  MoveL 2000 to (240.59, 49.33, 41.04) mm, rotated rx -180 ry 0 rz 180 deg; joints [-31.47, 47.148, -71.346, 33.863, 110.463, 13.203]
  Call Extruder(203.73378)
  MoveL 2001 to (240.64, 49.63, 41.04) mm, rotated rx -180 ry 0 rz 180 deg; joints [-31.612, 47.167, -71.344, 34.007, 110.413, 13.242]
  MoveL 2002 to (240.64, 49.63, 41.04) mm, rotated rx -180 ry 0 rz 180 deg; joints [-31.612, 47.167, -71.344, 34.007, 110.413, 13.242]
  Call Extruder(203.89480)
  MoveL 2003 to (240.69, 49.94, 41.04) mm, rotated rx 180 ry 0 rz 180 deg; joints [-31.755, 47.186, -71.343, 34.15, 110.364, 13.281]
  MoveL 2004 to (240.69, 49.94, 41.04) mm, rotated rx 180 ry 0 rz 180 deg; joints [-31.755, 47.186, -71.343, 34.15, 110.364, 13.281]
  Call Extruder(204.05509)
  MoveL 2005 to (240.74, 50.24, 41.04) mm, rotated rx 180 ry 0 rz 180 deg; joints [-31.895, 47.205, -71.341, 34.292, 110.314, 13.32]
  MoveL 2006 to (240.74, 50.24, 41.04) mm, rotated rx 180 ry 0 rz 180 deg; joints [-31.895, 47.205, -71.341, 34.292, 110.314, 13.32]
  Call Extruder(204.21465)
  MoveL 2007 to (240.78, 50.55, 41.04) mm, rotated rx 180 ry 0 rz 180 deg; joints [-32.036, 47.224, -71.34, 34.434, 110.265, 13.358]
  MoveL 2008 to (240.78, 50.55, 41.04) mm, rotated rx 180 ry 0 rz 180 deg; joints [-32.036, 47.224, -71.34, 34.434, 110.265, 13.358]
  Call Extruder(204.37349)
  MoveL 2009 to (240.83, 50.86, 41.04) mm, rotated rx -180 ry 0 rz 180 deg; joints [-32.176, 47.243, -71.338, 34.575, 110.215, 13.396]
  MoveL 2010 to (240.83, 50.86, 41.04) mm, rotated rx -180 ry 0 rz 180 deg; joints [-32.176, 47.243, -71.338, 34.575, 110.215, 13.396]
  Call Extruder(204.55216)
  MoveL 2011 to (240.88, 51.2, 41.04) mm, rotated rx 180 ry 0 rz -180 deg; joints [-32.337, 47.264, -71.336, 34.736, 110.159, 13.439]
  MoveL 2012 to (240.88, 51.2, 41.04) mm, rotated rx 180 ry 0 rz -180 deg; joints [-32.337, 47.264, -71.336, 34.736, 110.159, 13.439]
  Call Extruder(204.75060)
  MoveL 2013 to (240.92, 51.59, 41.04) mm, rotated rx -180 ry 0 rz 180 deg; joints [-32.518, 47.288, -71.334, 34.918, 110.096, 13.488]
  MoveL 2014 to (240.92, 51.59, 41.04) mm, rotated rx -180 ry 0 rz 180 deg; joints [-32.518, 47.288, -71.334, 34.918, 110.096, 13.488]
  Call Extruder(204.94818)
  MoveL 2015 to (240.97, 51.98, 41.04) mm, rotated rx 180 ry 0 rz 180 deg; joints [-32.697, 47.311, -71.332, 35.099, 110.034, 13.537]
  MoveL 2016 to (240.97, 51.98, 41.04) mm, rotated rx 180 ry 0 rz 180 deg; joints [-32.697, 47.311, -71.332, 35.099, 110.034, 13.537]
  Call Extruder(205.14488)
  MoveL 2017 to (241.02, 52.37, 41.04) mm, rotated rx -180 ry 0 rz 180 deg; joints [-32.876, 47.334, -71.33, 35.279, 109.971, 13.584]
  MoveL 2018 to (241.02, 52.37, 41.04) mm, rotated rx -180 ry 0 rz 180 deg; joints [-32.876, 47.334, -71.33, 35.279, 109.971, 13.584]
  Call Extruder(205.34072)
  MoveL 2019 to (241.06, 52.75, 41.04) mm, rotated rx 180 ry 0 rz 180 deg; joints [-33.055, 47.357, -71.328, 35.458, 109.908, 13.632]
  MoveL 2020 to (241.06, 52.75, 41.04) mm, rotated rx 180 ry 0 rz 180 deg; joints [-33.055, 47.357, -71.328, 35.458, 109.908, 13.632]
  Call Extruder(205.63616)
  MoveL 2021 to (241.11, 53.34, 41.04) mm, rotated rx -180 ry 0 rz 180 deg; joints [-33.331, 47.391, -71.325, 35.736, 109.813, 13.706]
  MoveL 2022 to (241.11, 53.34, 41.04) mm, rotated rx -180 ry 0 rz 180 deg; joints [-33.331, 47.391, -71.325, 35.736, 109.813, 13.706]
  Call Extruder(205.93027)
  MoveL 2023 to (241.16, 53.93, 41.04) mm, rotated rx 180 ry 0 rz 180 deg; joints [-33.606, 47.426, -71.322, 36.012, 109.717, 13.779]
  MoveL 2024 to (241.16, 53.93, 41.04) mm, rotated rx 180 ry 0 rz 180 deg; joints [-33.606, 47.426, -71.322, 36.012, 109.717, 13.779]
  Call Extruder(206.22304)
  MoveL 2025 to (241.2, 54.52, 41.04) mm, rotated rx -180 ry 0 rz 180 deg; joints [-33.878, 47.46, -71.319, 36.285, 109.622, 13.85]
  MoveL 2026 to (241.2, 54.52, 41.04) mm, rotated rx -180 ry 0 rz 180 deg; joints [-33.878, 47.46, -71.319, 36.285, 109.622, 13.85]
  Call Extruder(206.79649)
  MoveL 2027 to (241.25, 55.68, 41.04) mm, rotated rx 180 ry 0 rz 180 deg; joints [-34.425, 47.525, -71.313, 36.832, 109.434, 13.993]
  MoveL 2028 to (241.25, 55.68, 41.04) mm, rotated rx 180 ry 0 rz 180 deg; joints [-34.425, 47.525, -71.313, 36.832, 109.434, 13.993]
  Call Extruder(207.51032)
  MoveL 2029 to (241.29, 57.14, 41.04) mm, rotated rx 180 ry 0 rz 180 deg; joints [-35.104, 47.605, -71.305, 37.512, 109.198, 14.167]
  Call Extruder(249.57521)
  MoveL 2030 to (241.29, 142.86, 41.03) mm, rotated rx 180 ry 0 rz 180 deg; joints [-60.361, 53.167, -69.896, 61.414, 98.184, 14.641]
  Call Extruder(250.00364)
  MoveL 2031 to (241.27, 143.73, 41.04) mm, rotated rx -180 ry 0 rz 180 deg; joints [-60.516, 53.225, -69.87, 61.555, 98.105, 14.588]
  MoveL 2032 to (241.27, 143.73, 41.04) mm, rotated rx -180 ry 0 rz 180 deg; joints [-60.516, 53.225, -69.87, 61.555, 98.105, 14.588]
  Call Extruder(250.57709)
  MoveL 2033 to (241.23, 144.9, 41.04) mm, rotated rx 180 ry 0 rz 180 deg; joints [-60.726, 53.301, -69.836, 61.747, 97.999, 14.519]
  MoveL 2034 to (241.23, 144.9, 41.04) mm, rotated rx 180 ry 0 rz 180 deg; joints [-60.726, 53.301, -69.836, 61.747, 97.999, 14.519]
  Call Extruder(251.01142)
  MoveL 2035 to (241.18, 145.77, 41.04) mm, rotated rx 180 ry 0 rz 180 deg; joints [-60.887, 53.358, -69.81, 61.894, 97.92, 14.467]
  MoveL 2036 to (241.18, 145.77, 41.04) mm, rotated rx 180 ry 0 rz 180 deg; joints [-60.887, 53.358, -69.81, 61.894, 97.92, 14.467]
  Call Extruder(251.30553)
  MoveL 2037 to (241.13, 146.36, 41.04) mm, rotated rx -180 ry 0 rz 180 deg; joints [-61, 53.396, -69.793, 61.997, 97.866, 14.433]
  MoveL 2038 to (241.13, 146.36, 41.04) mm, rotated rx -180 ry 0 rz 180 deg; joints [-61, 53.396, -69.793, 61.997, 97.866, 14.433]
  Call Extruder(251.60097)
  MoveL 2039 to (241.09, 146.95, 41.04) mm, rotated rx -180 ry 0 rz 180 deg; joints [-61.111, 53.434, -69.775, 62.099, 97.813, 14.398]
  MoveL 2040 to (241.09, 146.95, 41.04) mm, rotated rx -180 ry 0 rz 180 deg; joints [-61.111, 53.434, -69.775, 62.099, 97.813, 14.398]
  Call Extruder(251.84723)
  MoveL 2041 to (241.04, 147.44, 41.04) mm, rotated rx 180 ry 0 rz 180 deg; joints [-61.205, 53.465, -69.761, 62.186, 97.768, 14.37]
  MoveL 2042 to (241.04, 147.44, 41.04) mm, rotated rx 180 ry 0 rz 180 deg; joints [-61.205, 53.465, -69.761, 62.186, 97.768, 14.37]
  Call Extruder(252.04393)
  MoveL 2043 to (240.99, 147.83, 41.04) mm, rotated rx 180 ry 0 rz 180 deg; joints [-61.282, 53.489, -69.75, 62.257, 97.732, 14.349]
  MoveL 2044 to (240.99, 147.83, 41.04) mm, rotated rx 180 ry 0 rz 180 deg; joints [-61.282, 53.489, -69.75, 62.257, 97.732, 14.349]
  Call Extruder(252.24151)
  MoveL 2045 to (240.95, 148.22, 41.04) mm, rotated rx -180 ry 0 rz 180 deg; joints [-61.359, 53.513, -69.738, 62.328, 97.697, 14.327]
  MoveL 2046 to (240.95, 148.22, 41.04) mm, rotated rx -180 ry 0 rz 180 deg; joints [-61.359, 53.513, -69.738, 62.328, 97.697, 14.327]
  Call Extruder(252.43995)
  MoveL 2047 to (240.9, 148.6, 41.04) mm, rotated rx -180 ry 0 rz 180 deg; joints [-61.436, 53.537, -69.727, 62.398, 97.661, 14.305]
  MoveL 2048 to (240.9, 148.6, 41.04) mm, rotated rx -180 ry 0 rz 180 deg; joints [-61.436, 53.537, -69.727, 62.398, 97.661, 14.305]
  Call Extruder(252.63926)
  MoveL 2049 to (240.86, 148.99, 41.04) mm, rotated rx 180 ry 0 rz 180 deg; joints [-61.512, 53.562, -69.715, 62.469, 97.626, 14.283]
  MoveL 2050 to (240.86, 148.99, 41.04) mm, rotated rx 180 ry 0 rz 180 deg; joints [-61.512, 53.562, -69.715, 62.469, 97.626, 14.283]
  Call Extruder(252.79809)
  MoveL 2051 to (240.81, 149.3, 41.04) mm, rotated rx -180 ry 0 rz 180 deg; joints [-61.575, 53.58, -69.707, 62.527, 97.597, 14.266]
  MoveL 2052 to (240.81, 149.3, 41.04) mm, rotated rx -180 ry 0 rz 180 deg; joints [-61.575, 53.58, -69.707, 62.527, 97.597, 14.266]
  Call Extruder(252.95765)
  MoveL 2053 to (240.76, 149.6, 41.04) mm, rotated rx 180 ry 0 rz 180 deg; joints [-61.639, 53.599, -69.698, 62.586, 97.569, 14.25]
  MoveL 2054 to (240.76, 149.6, 41.04) mm, rotated rx 180 ry 0 rz 180 deg; joints [-61.639, 53.599, -69.698, 62.586, 97.569, 14.25]
  Call Extruder(253.11794)
  MoveL 2055 to (240.71, 149.91, 41.04) mm, rotated rx -180 ry 0 rz 180 deg; joints [-61.702, 53.618, -69.689, 62.645, 97.541, 14.233]
  MoveL 2056 to (240.71, 149.91, 41.04) mm, rotated rx -180 ry 0 rz 180 deg; joints [-61.702, 53.618, -69.689, 62.645, 97.541, 14.233]
  Call Extruder(253.27896)
  MoveL 2057 to (240.66, 150.21, 41.04) mm, rotated rx 180 ry 0 rz -180 deg; joints [-61.765, 53.636, -69.68, 62.703, 97.513, 14.217]
  MoveL 2058 to (240.66, 150.21, 41.04) mm, rotated rx 180 ry 0 rz -180 deg; joints [-61.765, 53.636, -69.68, 62.703, 97.513, 14.217]
  Call Extruder(253.44070)
  MoveL 2059 to (240.61, 150.52, 41.04) mm, rotated rx -180 ry 0 rz 180 deg; joints [-61.828, 53.655, -69.671, 62.761, 97.485, 14.2]
  MoveL 2060 to (240.61, 150.52, 41.04) mm, rotated rx -180 ry 0 rz 180 deg; joints [-61.828, 53.655, -69.671, 62.761, 97.485, 14.2]
  Call Extruder(253.60317)
  MoveL 2061 to (240.56, 150.83, 41.04) mm, rotated rx -180 ry 0 rz 180 deg; joints [-61.891, 53.674, -69.662, 62.82, 97.456, 14.183]
  MoveL 2062 to (240.56, 150.83, 41.04) mm, rotated rx -180 ry 0 rz 180 deg; joints [-61.891, 53.674, -69.662, 62.82, 97.456, 14.183]
  Call Extruder(253.73710)
  MoveL 2063 to (240.52, 151.08, 41.04) mm, rotated rx -180 ry 0 rz 180 deg; joints [-61.944, 53.689, -69.654, 62.87, 97.433, 14.17]
  MoveL 2064 to (240.52, 151.08, 41.04) mm, rotated rx -180 ry 0 rz 180 deg; joints [-61.944, 53.689, -69.654, 62.87, 97.433, 14.17]
  Call Extruder(253.87164)
  MoveL 2065 to (240.47, 151.32, 41.04) mm, rotated rx -180 ry 0 rz 180 deg; joints [-61.998, 53.703, -69.647, 62.92, 97.41, 14.157]
  MoveL 2066 to (240.47, 151.32, 41.04) mm, rotated rx -180 ry 0 rz 180 deg; joints [-61.998, 53.703, -69.647, 62.92, 97.41, 14.157]
  Call Extruder(254.00678)
  MoveL 2067 to (240.42, 151.57, 41.04) mm, rotated rx -180 ry 0 rz 180 deg; joints [-62.052, 53.718, -69.64, 62.97, 97.387, 14.144]
  MoveL 2068 to (240.42, 151.57, 41.04) mm, rotated rx -180 ry 0 rz 180 deg; joints [-62.052, 53.718, -69.64, 62.97, 97.387, 14.144]
  Call Extruder(254.14254)
  MoveL 2069 to (240.37, 151.82, 41.04) mm, rotated rx -180 ry 0 rz 180 deg; joints [-62.105, 53.733, -69.633, 63.019, 97.364, 14.131]
  MoveL 2070 to (240.37, 151.82, 41.04) mm, rotated rx -180 ry 0 rz 180 deg; joints [-62.105, 53.733, -69.633, 63.019, 97.364, 14.131]
  Call Extruder(254.27891)
  MoveL 2071 to (240.32, 152.07, 41.04) mm, rotated rx 180 ry 0 rz 180 deg; joints [-62.159, 53.748, -69.625, 63.069, 97.341, 14.118]
  MoveL 2072 to (240.32, 152.07, 41.04) mm, rotated rx 180 ry 0 rz 180 deg; joints [-62.159, 53.748, -69.625, 63.069, 97.341, 14.118]
  Call Extruder(254.41589)
  MoveL 2073 to (240.27, 152.32, 41.04) mm, rotated rx -180 ry 0 rz 180 deg; joints [-62.212, 53.763, -69.618, 63.119, 97.318, 14.104]
  MoveL 2074 to (240.27, 152.32, 41.04) mm, rotated rx -180 ry 0 rz 180 deg; joints [-62.212, 53.763, -69.618, 63.119, 97.318, 14.104]
  Call Extruder(254.55347)
  MoveL 2075 to (240.22, 152.57, 41.04) mm, rotated rx -180 ry 0 rz 180 deg; joints [-62.265, 53.778, -69.611, 63.168, 97.295, 14.091]
  MoveL 2076 to (240.22, 152.57, 41.04) mm, rotated rx -180 ry 0 rz 180 deg; joints [-62.265, 53.778, -69.611, 63.168, 97.295, 14.091]
  Call Extruder(254.66717)
  MoveL 2077 to (240.17, 152.77, 41.04) mm, rotated rx -180 ry 0 rz -180 deg; joints [-62.31, 53.79, -69.605, 63.21, 97.276, 14.08]
  MoveL 2078 to (240.17, 152.77, 41.04) mm, rotated rx -180 ry 0 rz -180 deg; joints [-62.31, 53.79, -69.605, 63.21, 97.276, 14.08]
  Call Extruder(254.78132)
  MoveL 2079 to (240.13, 152.98, 41.04) mm, rotated rx -180 ry 0 rz -180 deg; joints [-62.355, 53.802, -69.599, 63.251, 97.257, 14.07]
  MoveL 2080 to (240.13, 152.98, 41.04) mm, rotated rx -180 ry 0 rz -180 deg; joints [-62.355, 53.802, -69.599, 63.251, 97.257, 14.07]
  Call Extruder(254.89592)
  MoveL 2081 to (240.08, 153.18, 41.04) mm, rotated rx 180 ry 0 rz 180 deg; joints [-62.399, 53.814, -69.593, 63.293, 97.238, 14.059]
  MoveL 2082 to (240.08, 153.18, 41.04) mm, rotated rx 180 ry 0 rz 180 deg; joints [-62.399, 53.814, -69.593, 63.293, 97.238, 14.059]
  Call Extruder(255.01098)
  MoveL 2083 to (240.04, 153.39, 41.04) mm, rotated rx 180 ry 0 rz -180 deg; joints [-62.444, 53.826, -69.587, 63.334, 97.219, 14.048]
  MoveL 2084 to (240.04, 153.39, 41.04) mm, rotated rx 180 ry 0 rz -180 deg; joints [-62.444, 53.826, -69.587, 63.334, 97.219, 14.048]
  Call Extruder(255.13320)
  MoveL 2085 to (239.98, 153.6, 41.03) mm, rotated rx -180 ry 0 rz 180 deg; joints [-62.493, 53.838, -69.581, 63.38, 97.199, 14.037]
  MoveL 2086 to (239.98, 153.6, 41.03) mm, rotated rx -180 ry 0 rz 180 deg; joints [-62.493, 53.838, -69.581, 63.38, 97.199, 14.037]
  Call Extruder(255.26286)
  MoveL 2087 to (239.92, 153.82, 41.04) mm, rotated rx -180 ry 0 rz 180 deg; joints [-62.547, 53.851, -69.574, 63.431, 97.177, 14.027]
  MoveL 2088 to (239.92, 153.82, 41.04) mm, rotated rx -180 ry 0 rz 180 deg; joints [-62.547, 53.851, -69.574, 63.431, 97.177, 14.027]
  Call Extruder(255.39309)
  MoveL 2089 to (239.85, 154.05, 41.04) mm, rotated rx -180 ry 0 rz 180 deg; joints [-62.601, 53.863, -69.568, 63.481, 97.156, 14.017]
  MoveL 2090 to (239.85, 154.05, 41.04) mm, rotated rx -180 ry 0 rz 180 deg; joints [-62.601, 53.863, -69.568, 63.481, 97.156, 14.017]
  Call Extruder(255.52388)
  MoveL 2091 to (239.78, 154.27, 41.04) mm, rotated rx -180 ry 0 rz -180 deg; joints [-62.654, 53.876, -69.562, 63.532, 97.134, 14.006]
  MoveL 2092 to (239.78, 154.27, 41.04) mm, rotated rx -180 ry 0 rz -180 deg; joints [-62.654, 53.876, -69.562, 63.532, 97.134, 14.006]
  Call Extruder(255.65523)
  MoveL 2093 to (239.71, 154.49, 41.04) mm, rotated rx -180 ry 0 rz 180 deg; joints [-62.708, 53.888, -69.556, 63.582, 97.113, 13.996]
  MoveL 2094 to (239.71, 154.49, 41.04) mm, rotated rx -180 ry 0 rz 180 deg; joints [-62.708, 53.888, -69.556, 63.582, 97.113, 13.996]
  Call Extruder(255.76713)
  MoveL 2095 to (239.65, 154.68, 41.04) mm, rotated rx 180 ry 0 rz 180 deg; joints [-62.754, 53.899, -69.55, 63.626, 97.095, 13.987]
  MoveL 2096 to (239.65, 154.68, 41.04) mm, rotated rx 180 ry 0 rz 180 deg; joints [-62.754, 53.899, -69.55, 63.626, 97.095, 13.987]
  Call Extruder(255.87948)
  MoveL 2097 to (239.59, 154.87, 41.04) mm, rotated rx -180 ry 0 rz -180 deg; joints [-62.801, 53.909, -69.545, 63.669, 97.076, 13.978]
  MoveL 2098 to (239.59, 154.87, 41.04) mm, rotated rx -180 ry 0 rz -180 deg; joints [-62.801, 53.909, -69.545, 63.669, 97.076, 13.978]
  Call Extruder(255.99227)
  MoveL 2099 to (239.53, 155.06, 41.04) mm, rotated rx -180 ry 0 rz 180 deg; joints [-62.847, 53.92, -69.54, 63.713, 97.058, 13.97]
  MoveL 2100 to (239.53, 155.06, 41.04) mm, rotated rx -180 ry 0 rz 180 deg; joints [-62.847, 53.92, -69.54, 63.713, 97.058, 13.97]
  Call Extruder(256.10550)
  MoveL 2101 to (239.47, 155.25, 41.04) mm, rotated rx 180 ry 0 rz 180 deg; joints [-62.893, 53.93, -69.534, 63.756, 97.04, 13.961]
  MoveL 2102 to (239.47, 155.25, 41.04) mm, rotated rx 180 ry 0 rz 180 deg; joints [-62.893, 53.93, -69.534, 63.756, 97.04, 13.961]
  Call Extruder(256.21918)
  MoveL 2103 to (239.41, 155.44, 41.04) mm, rotated rx -180 ry 0 rz 180 deg; joints [-62.939, 53.941, -69.529, 63.8, 97.022, 13.952]
  MoveL 2104 to (239.41, 155.44, 41.04) mm, rotated rx -180 ry 0 rz 180 deg; joints [-62.939, 53.941, -69.529, 63.8, 97.022, 13.952]
  Call Extruder(256.40114)
  MoveL 2105 to (239.29, 155.73, 41.04) mm, rotated rx 180 ry 0 rz 180 deg; joints [-63.018, 53.956, -69.521, 63.874, 96.993, 13.941]
  MoveL 2106 to (239.29, 155.73, 41.04) mm, rotated rx 180 ry 0 rz 180 deg; joints [-63.018, 53.956, -69.521, 63.874, 96.993, 13.941]
  Call Extruder(256.58386)
  MoveL 2107 to (239.16, 156.02, 41.04) mm, rotated rx -180 ry 0 rz 180 deg; joints [-63.097, 53.971, -69.513, 63.948, 96.964, 13.929]
  MoveL 2108 to (239.16, 156.02, 41.04) mm, rotated rx -180 ry 0 rz 180 deg; joints [-63.097, 53.971, -69.513, 63.948, 96.964, 13.929]
  Call Extruder(256.75428)
  MoveL 2109 to (239.05, 156.29, 41.04) mm, rotated rx 180 ry 0 rz 180 deg; joints [-63.17, 53.985, -69.506, 64.018, 96.937, 13.919]
  MoveL 2110 to (239.05, 156.29, 41.04) mm, rotated rx 180 ry 0 rz 180 deg; joints [-63.17, 53.985, -69.506, 64.018, 96.937, 13.919]
  Call Extruder(256.91229)
  MoveL 2111 to (238.94, 156.54, 41.04) mm, rotated rx 180 ry 0 rz 180 deg; joints [-63.238, 53.998, -69.5, 64.082, 96.912, 13.909]
  MoveL 2112 to (238.94, 156.54, 41.04) mm, rotated rx 180 ry 0 rz 180 deg; joints [-63.238, 53.998, -69.5, 64.082, 96.912, 13.909]
  Call Extruder(257.07091)
  MoveL 2113 to (238.84, 156.79, 41.04) mm, rotated rx 180 ry 0 rz 180 deg; joints [-63.306, 54.011, -69.493, 64.146, 96.887, 13.899]
  MoveL 2114 to (238.84, 156.79, 41.04) mm, rotated rx 180 ry 0 rz 180 deg; joints [-63.306, 54.011, -69.493, 64.146, 96.887, 13.899]
  Call Extruder(257.27708)
  MoveL 2115 to (238.66, 157.09, 41.04) mm, rotated rx 180 ry 0 rz -180 deg; joints [-63.401, 54.026, -69.485, 64.237, 96.854, 13.89]
  MoveL 2116 to (238.66, 157.09, 41.04) mm, rotated rx 180 ry 0 rz -180 deg; joints [-63.401, 54.026, -69.485, 64.237, 96.854, 13.89]
  Call Extruder(257.48403)
  MoveL 2117 to (238.49, 157.4, 41.03) mm, rotated rx 180 ry 0 rz 180 deg; joints [-63.497, 54.04, -69.478, 64.328, 96.822, 13.882]
  MoveL 2118 to (238.49, 157.4, 41.03) mm, rotated rx 180 ry 0 rz 180 deg; joints [-63.497, 54.04, -69.478, 64.328, 96.822, 13.882]
  Call Extruder(257.69175)
  MoveL 2119 to (238.31, 157.7, 41.04) mm, rotated rx -180 ry 0 rz 180 deg; joints [-63.592, 54.055, -69.47, 64.419, 96.79, 13.873]
  MoveL 2120 to (238.31, 157.7, 41.04) mm, rotated rx -180 ry 0 rz 180 deg; joints [-63.592, 54.055, -69.47, 64.419, 96.79, 13.873]
  Call Extruder(257.90025)
  MoveL 2121 to (238.13, 158.01, 41.04) mm, rotated rx -180 ry 0 rz 180 deg; joints [-63.687, 54.069, -69.463, 64.51, 96.758, 13.864]
  MoveL 2122 to (238.13, 158.01, 41.04) mm, rotated rx -180 ry 0 rz 180 deg; joints [-63.687, 54.069, -69.463, 64.51, 96.758, 13.864]
  Call Extruder(258.07978)
  MoveL 2123 to (237.96, 158.25, 41.04) mm, rotated rx -180 ry 0 rz 180 deg; joints [-63.774, 54.08, -69.457, 64.593, 96.73, 13.859]
  MoveL 2124 to (237.96, 158.25, 41.04) mm, rotated rx -180 ry 0 rz 180 deg; joints [-63.774, 54.08, -69.457, 64.593, 96.73, 13.859]
  Call Extruder(258.41320)
  MoveL 2125 to (237.63, 158.7, 41.04) mm, rotated rx 180 ry 0 rz -180 deg; joints [-63.934, 54.099, -69.447, 64.746, 96.679, 13.851]
  MoveL 2126 to (237.63, 158.7, 41.04) mm, rotated rx 180 ry 0 rz -180 deg; joints [-63.934, 54.099, -69.447, 64.746, 96.679, 13.851]
  Call Extruder(258.74780)
  MoveL 2127 to (237.3, 159.15, 41.04) mm, rotated rx 180 ry 0 rz 180 deg; joints [-64.094, 54.118, -69.437, 64.899, 96.628, 13.842]
  Call Extruder(259.57575)
  MoveL 2128 to (236.39, 160.19, 41.04) mm, rotated rx -180 ry 0 rz 180 deg; joints [-64.505, 54.158, -69.416, 65.294, 96.504, 13.832]
  Call Extruder(260.40368)
  MoveL 2129 to (235.35, 161.1, 41.04) mm, rotated rx 180 ry 0 rz -180 deg; joints [-64.933, 54.186, -69.401, 65.708, 96.384, 13.839]
  Call Extruder(260.57099)
  MoveL 2130 to (235.13, 161.27, 41.04) mm, rotated rx -180 ry 0 rz 180 deg; joints [-65.021, 54.19, -69.399, 65.794, 96.36, 13.844]
  MoveL 2131 to (235.13, 161.27, 41.04) mm, rotated rx -180 ry 0 rz 180 deg; joints [-65.021, 54.19, -69.399, 65.794, 96.36, 13.844]
  Call Extruder(260.90442)
  MoveL 2132 to (234.68, 161.59, 41.04) mm, rotated rx -180 ry 0 rz 180 deg; joints [-65.197, 54.198, -69.395, 65.965, 96.313, 13.851]
  MoveL 2133 to (234.68, 161.59, 41.04) mm, rotated rx -180 ry 0 rz 180 deg; joints [-65.197, 54.198, -69.395, 65.965, 96.313, 13.851]
  Call Extruder(261.23666)
  MoveL 2134 to (234.22, 161.92, 41.04) mm, rotated rx -180 ry 0 rz 180 deg; joints [-65.374, 54.206, -69.39, 66.136, 96.266, 13.859]
  MoveL 2135 to (234.22, 161.92, 41.04) mm, rotated rx -180 ry 0 rz 180 deg; joints [-65.374, 54.206, -69.39, 66.136, 96.266, 13.859]
  Call Extruder(261.35431)
  MoveL 2136 to (234.05, 162.02, 41.04) mm, rotated rx -180 ry 0 rz 180 deg; joints [-65.437, 54.208, -69.39, 66.197, 96.25, 13.864]
  MoveL 2137 to (234.05, 162.02, 41.04) mm, rotated rx -180 ry 0 rz 180 deg; joints [-65.437, 54.208, -69.39, 66.197, 96.25, 13.864]
  Call Extruder(261.56204)
  MoveL 2138 to (233.75, 162.2, 41.04) mm, rotated rx 180 ry 0 rz 180 deg; joints [-65.549, 54.21, -69.388, 66.307, 96.221, 13.872]
  MoveL 2139 to (233.75, 162.2, 41.04) mm, rotated rx 180 ry 0 rz 180 deg; joints [-65.549, 54.21, -69.388, 66.307, 96.221, 13.872]
  Call Extruder(261.76899)
  MoveL 2140 to (233.45, 162.37, 41.04) mm, rotated rx -180 ry 0 rz 180 deg; joints [-65.662, 54.213, -69.387, 66.416, 96.193, 13.88]
  MoveL 2141 to (233.45, 162.37, 41.04) mm, rotated rx -180 ry 0 rz 180 deg; joints [-65.662, 54.213, -69.387, 66.416, 96.193, 13.88]
  Call Extruder(261.97516)
  MoveL 2142 to (233.14, 162.55, 41.04) mm, rotated rx -180 ry 0 rz 180 deg; joints [-65.774, 54.215, -69.386, 66.525, 96.164, 13.888]
  MoveL 2143 to (233.14, 162.55, 41.04) mm, rotated rx -180 ry 0 rz 180 deg; joints [-65.774, 54.215, -69.386, 66.525, 96.164, 13.888]
  Call Extruder(262.15683)
  MoveL 2144 to (232.87, 162.69, 41.04) mm, rotated rx 180 ry 0 rz -180 deg; joints [-65.874, 54.216, -69.385, 66.623, 96.14, 13.897]
  MoveL 2145 to (232.87, 162.69, 41.04) mm, rotated rx 180 ry 0 rz -180 deg; joints [-65.874, 54.216, -69.385, 66.623, 96.14, 13.897]
  Call Extruder(262.31480)
  MoveL 2146 to (232.62, 162.8, 41.03) mm, rotated rx -180 ry 0 rz 180 deg; joints [-65.961, 54.216, -69.385, 66.708, 96.119, 13.907]
  MoveL 2147 to (232.62, 162.8, 41.03) mm, rotated rx -180 ry 0 rz 180 deg; joints [-65.961, 54.216, -69.385, 66.708, 96.119, 13.907]
  Call Extruder(262.47217)
  MoveL 2148 to (232.37, 162.9, 41.04) mm, rotated rx -180 ry 0 rz 180 deg; joints [-66.048, 54.216, -69.385, 66.793, 96.098, 13.916]
  MoveL 2149 to (232.37, 162.9, 41.04) mm, rotated rx -180 ry 0 rz 180 deg; joints [-66.048, 54.216, -69.385, 66.793, 96.098, 13.916]
  Call Extruder(262.65491)
  MoveL 2150 to (232.07, 163.03, 41.04) mm, rotated rx 180 ry 0 rz -180 deg; joints [-66.149, 54.215, -69.386, 66.892, 96.074, 13.928]
  MoveL 2151 to (232.07, 163.03, 41.04) mm, rotated rx 180 ry 0 rz -180 deg; joints [-66.149, 54.215, -69.386, 66.892, 96.074, 13.928]
  Call Extruder(262.83690)
  MoveL 2152 to (231.78, 163.15, 41.04) mm, rotated rx -180 ry 0 rz 180 deg; joints [-66.251, 54.215, -69.386, 66.991, 96.05, 13.939]
  MoveL 2153 to (231.78, 163.15, 41.04) mm, rotated rx -180 ry 0 rz 180 deg; joints [-66.251, 54.215, -69.386, 66.991, 96.05, 13.939]
  Call Extruder(262.98424)
  MoveL 2154 to (231.54, 163.24, 41.04) mm, rotated rx -180 ry 0 rz 180 deg; joints [-66.333, 54.214, -69.386, 67.072, 96.031, 13.949]
  MoveL 2155 to (231.54, 163.24, 41.04) mm, rotated rx -180 ry 0 rz 180 deg; joints [-66.333, 54.214, -69.386, 67.072, 96.031, 13.949]
  Call Extruder(263.09746)
  MoveL 2156 to (231.35, 163.3, 41.04) mm, rotated rx 180 ry 0 rz -180 deg; joints [-66.397, 54.212, -69.387, 67.134, 96.016, 13.957]
  MoveL 2157 to (231.35, 163.3, 41.04) mm, rotated rx 180 ry 0 rz -180 deg; joints [-66.397, 54.212, -69.387, 67.134, 96.016, 13.957]
  Call Extruder(263.21024)
  MoveL 2158 to (231.17, 163.36, 41.04) mm, rotated rx -180 ry 0 rz 180 deg; joints [-66.46, 54.211, -69.388, 67.196, 96.002, 13.966]
  MoveL 2159 to (231.17, 163.36, 41.04) mm, rotated rx -180 ry 0 rz 180 deg; joints [-66.46, 54.211, -69.388, 67.196, 96.002, 13.966]
  Call Extruder(263.32257)
  MoveL 2160 to (230.98, 163.42, 41.04) mm, rotated rx 180 ry 0 rz 180 deg; joints [-66.524, 54.21, -69.389, 67.258, 95.987, 13.974]
  MoveL 2161 to (230.98, 163.42, 41.04) mm, rotated rx 180 ry 0 rz 180 deg; joints [-66.524, 54.21, -69.389, 67.258, 95.987, 13.974]
  Call Extruder(263.43446)
  MoveL 2162 to (230.79, 163.48, 41.04) mm, rotated rx 180 ry 0 rz -180 deg; joints [-66.587, 54.208, -69.389, 67.32, 95.973, 13.982]
  MoveL 2163 to (230.79, 163.48, 41.04) mm, rotated rx 180 ry 0 rz -180 deg; joints [-66.587, 54.208, -69.389, 67.32, 95.973, 13.982]
  Call Extruder(263.55586)
  MoveL 2164 to (230.58, 163.55, 41.04) mm, rotated rx -180 ry 0 rz 180 deg; joints [-66.656, 54.207, -69.39, 67.388, 95.957, 13.992]
  MoveL 2165 to (230.58, 163.55, 41.04) mm, rotated rx -180 ry 0 rz 180 deg; joints [-66.656, 54.207, -69.39, 67.388, 95.957, 13.992]
  Call Extruder(263.68667)
  MoveL 2166 to (230.36, 163.62, 41.04) mm, rotated rx -180 ry 0 rz 180 deg; joints [-66.731, 54.205, -69.391, 67.461, 95.94, 14.002]
  MoveL 2167 to (230.36, 163.62, 41.04) mm, rotated rx -180 ry 0 rz 180 deg; joints [-66.731, 54.205, -69.391, 67.461, 95.94, 14.002]
  Call Extruder(263.81692)
  MoveL 2168 to (230.14, 163.68, 41.04) mm, rotated rx 180 ry 0 rz 180 deg; joints [-66.805, 54.203, -69.392, 67.534, 95.923, 14.012]
  MoveL 2169 to (230.14, 163.68, 41.04) mm, rotated rx 180 ry 0 rz 180 deg; joints [-66.805, 54.203, -69.392, 67.534, 95.923, 14.012]
  Call Extruder(263.94661)
  MoveL 2170 to (229.91, 163.75, 41.04) mm, rotated rx -180 ry 0 rz -180 deg; joints [-66.88, 54.201, -69.393, 67.607, 95.906, 14.023]
  MoveL 2171 to (229.91, 163.75, 41.04) mm, rotated rx -180 ry 0 rz -180 deg; joints [-66.88, 54.201, -69.393, 67.607, 95.906, 14.023]
  Call Extruder(264.07572)
  MoveL 2172 to (229.69, 163.82, 41.04) mm, rotated rx -180 ry 0 rz -180 deg; joints [-66.955, 54.199, -69.394, 67.68, 95.889, 14.033]
  MoveL 2173 to (229.69, 163.82, 41.04) mm, rotated rx -180 ry 0 rz -180 deg; joints [-66.955, 54.199, -69.394, 67.68, 95.889, 14.033]
  Call Extruder(264.19080)
  MoveL 2174 to (229.48, 163.86, 41.04) mm, rotated rx 180 ry 0 rz 180 deg; joints [-67.021, 54.196, -69.396, 67.745, 95.875, 14.043]
  MoveL 2175 to (229.48, 163.86, 41.04) mm, rotated rx 180 ry 0 rz 180 deg; joints [-67.021, 54.196, -69.396, 67.745, 95.875, 14.043]
  Call Extruder(264.30542)
  MoveL 2176 to (229.28, 163.91, 41.04) mm, rotated rx -180 ry 0 rz 180 deg; joints [-67.087, 54.193, -69.397, 67.81, 95.86, 14.054]
  MoveL 2177 to (229.28, 163.91, 41.04) mm, rotated rx -180 ry 0 rz 180 deg; joints [-67.087, 54.193, -69.397, 67.81, 95.86, 14.054]
  Call Extruder(264.41959)
  MoveL 2178 to (229.08, 163.95, 41.04) mm, rotated rx -180 ry 0 rz 180 deg; joints [-67.153, 54.19, -69.399, 67.875, 95.846, 14.065]
  MoveL 2179 to (229.08, 163.95, 41.04) mm, rotated rx -180 ry 0 rz 180 deg; joints [-67.153, 54.19, -69.399, 67.875, 95.846, 14.065]
  Call Extruder(264.53331)
  MoveL 2180 to (228.87, 164, 41.04) mm, rotated rx -180 ry 0 rz 180 deg; joints [-67.22, 54.188, -69.4, 67.94, 95.832, 14.075]
  MoveL 2181 to (228.87, 164, 41.04) mm, rotated rx -180 ry 0 rz 180 deg; joints [-67.22, 54.188, -69.4, 67.94, 95.832, 14.075]
  Call Extruder(264.65873)
  MoveL 2182 to (228.64, 164.04, 41.04) mm, rotated rx -180 ry 0 rz -180 deg; joints [-67.293, 54.184, -69.402, 68.012, 95.816, 14.087]
  MoveL 2183 to (228.64, 164.04, 41.04) mm, rotated rx -180 ry 0 rz -180 deg; joints [-67.293, 54.184, -69.402, 68.012, 95.816, 14.087]
  Call Extruder(264.79570)
  MoveL 2184 to (228.4, 164.09, 41.04) mm, rotated rx -180 ry 0 rz -180 deg; joints [-67.373, 54.181, -69.404, 68.091, 95.798, 14.1]
  MoveL 2185 to (228.4, 164.09, 41.04) mm, rotated rx -180 ry 0 rz -180 deg; joints [-67.373, 54.181, -69.404, 68.091, 95.798, 14.1]
  Call Extruder(264.93207)
  MoveL 2186 to (228.15, 164.14, 41.04) mm, rotated rx -180 ry 0 rz 180 deg; joints [-67.453, 54.177, -69.406, 68.17, 95.781, 14.114]
  MoveL 2187 to (228.15, 164.14, 41.04) mm, rotated rx -180 ry 0 rz 180 deg; joints [-67.453, 54.177, -69.406, 68.17, 95.781, 14.114]
  Call Extruder(265.06783)
  MoveL 2188 to (227.9, 164.19, 41.04) mm, rotated rx 180 ry 0 rz 180 deg; joints [-67.534, 54.173, -69.408, 68.249, 95.763, 14.127]
  MoveL 2189 to (227.9, 164.19, 41.04) mm, rotated rx 180 ry 0 rz 180 deg; joints [-67.534, 54.173, -69.408, 68.249, 95.763, 14.127]
  Call Extruder(265.20298)
  MoveL 2190 to (227.65, 164.24, 41.03) mm, rotated rx 180 ry 0 rz 180 deg; joints [-67.614, 54.17, -69.41, 68.327, 95.746, 14.14]
  MoveL 2191 to (227.65, 164.24, 41.03) mm, rotated rx 180 ry 0 rz 180 deg; joints [-67.614, 54.17, -69.41, 68.327, 95.746, 14.14]
  Call Extruder(265.33751)
  MoveL 2192 to (227.4, 164.29, 41.04) mm, rotated rx 180 ry 0 rz 180 deg; joints [-67.695, 54.166, -69.412, 68.406, 95.728, 14.153]
  MoveL 2193 to (227.4, 164.29, 41.04) mm, rotated rx 180 ry 0 rz 180 deg; joints [-67.695, 54.166, -69.412, 68.406, 95.728, 14.153]
  Call Extruder(265.47144)
  MoveL 2194 to (227.15, 164.34, 41.04) mm, rotated rx 180 ry 0 rz 180 deg; joints [-67.775, 54.162, -69.414, 68.485, 95.71, 14.166]
  MoveL 2195 to (227.15, 164.34, 41.04) mm, rotated rx 180 ry 0 rz 180 deg; joints [-67.775, 54.162, -69.414, 68.485, 95.71, 14.166]
  Call Extruder(265.61931)
  MoveL 2196 to (226.87, 164.39, 41.04) mm, rotated rx -180 ry 0 rz 180 deg; joints [-67.864, 54.158, -69.416, 68.572, 95.691, 14.181]
  MoveL 2197 to (226.87, 164.39, 41.04) mm, rotated rx -180 ry 0 rz 180 deg; joints [-67.864, 54.158, -69.416, 68.572, 95.691, 14.181]
  Call Extruder(265.78105)
  MoveL 2198 to (226.57, 164.44, 41.04) mm, rotated rx -180 ry 0 rz -180 deg; joints [-67.961, 54.153, -69.419, 68.668, 95.67, 14.197]
  MoveL 2199 to (226.57, 164.44, 41.04) mm, rotated rx -180 ry 0 rz -180 deg; joints [-67.961, 54.153, -69.419, 68.668, 95.67, 14.197]
  Call Extruder(265.94206)
  MoveL 2200 to (226.26, 164.49, 41.04) mm, rotated rx 180 ry 0 rz 180 deg; joints [-68.059, 54.148, -69.422, 68.764, 95.649, 14.214]
  MoveL 2201 to (226.26, 164.49, 41.04) mm, rotated rx 180 ry 0 rz 180 deg; joints [-68.059, 54.148, -69.422, 68.764, 95.649, 14.214]
  Call Extruder(266.10234)
  MoveL 2202 to (225.96, 164.53, 41.04) mm, rotated rx 180 ry 0 rz 180 deg; joints [-68.156, 54.143, -69.424, 68.859, 95.628, 14.231]
  MoveL 2203 to (225.96, 164.53, 41.04) mm, rotated rx 180 ry 0 rz 180 deg; joints [-68.156, 54.143, -69.424, 68.859, 95.628, 14.231]
  Call Extruder(266.26190)
  MoveL 2204 to (225.65, 164.58, 41.04) mm, rotated rx 180 ry 0 rz 180 deg; joints [-68.254, 54.137, -69.427, 68.955, 95.607, 14.247]
  MoveL 2205 to (225.65, 164.58, 41.04) mm, rotated rx 180 ry 0 rz 180 deg; joints [-68.254, 54.137, -69.427, 68.955, 95.607, 14.247]
  Call Extruder(266.42073)
  MoveL 2206 to (225.34, 164.63, 41.04) mm, rotated rx -180 ry 0 rz 180 deg; joints [-68.351, 54.132, -69.43, 69.051, 95.585, 14.264]
  MoveL 2207 to (225.34, 164.63, 41.04) mm, rotated rx -180 ry 0 rz 180 deg; joints [-68.351, 54.132, -69.43, 69.051, 95.585, 14.264]
  Call Extruder(266.59940)
  MoveL 2208 to (225, 164.68, 41.04) mm, rotated rx 180 ry 0 rz 180 deg; joints [-68.461, 54.126, -69.433, 69.159, 95.562, 14.283]
  MoveL 2209 to (225, 164.68, 41.04) mm, rotated rx 180 ry 0 rz 180 deg; joints [-68.461, 54.126, -69.433, 69.159, 95.562, 14.283]
  Call Extruder(266.79784)
  MoveL 2210 to (224.61, 164.73, 41.04) mm, rotated rx -180 ry 0 rz 180 deg; joints [-68.583, 54.119, -69.437, 69.279, 95.535, 14.305]
  MoveL 2211 to (224.61, 164.73, 41.04) mm, rotated rx -180 ry 0 rz 180 deg; joints [-68.583, 54.119, -69.437, 69.279, 95.535, 14.305]
  Call Extruder(266.99542)
  MoveL 2212 to (224.22, 164.77, 41.04) mm, rotated rx 180 ry 0 rz 180 deg; joints [-68.706, 54.112, -69.441, 69.399, 95.509, 14.327]
  MoveL 2213 to (224.22, 164.77, 41.04) mm, rotated rx 180 ry 0 rz 180 deg; joints [-68.706, 54.112, -69.441, 69.399, 95.509, 14.327]
  Call Extruder(267.19212)
  MoveL 2214 to (223.83, 164.82, 41.04) mm, rotated rx 180 ry 0 rz 180 deg; joints [-68.828, 54.104, -69.444, 69.519, 95.483, 14.349]
  MoveL 2215 to (223.83, 164.82, 41.04) mm, rotated rx 180 ry 0 rz 180 deg; joints [-68.828, 54.104, -69.444, 69.519, 95.483, 14.349]
  Call Extruder(267.38796)
  MoveL 2216 to (223.45, 164.86, 41.04) mm, rotated rx -180 ry 0 rz 180 deg; joints [-68.951, 54.097, -69.448, 69.639, 95.456, 14.371]
  MoveL 2217 to (223.45, 164.86, 41.04) mm, rotated rx -180 ry 0 rz 180 deg; joints [-68.951, 54.097, -69.448, 69.639, 95.456, 14.371]
  Call Extruder(267.68332)
  MoveL 2218 to (222.86, 164.91, 41.04) mm, rotated rx 180 ry 0 rz 180 deg; joints [-69.135, 54.085, -69.455, 69.82, 95.417, 14.405]
  MoveL 2219 to (222.86, 164.91, 41.04) mm, rotated rx 180 ry 0 rz 180 deg; joints [-69.135, 54.085, -69.455, 69.82, 95.417, 14.405]
  Call Extruder(267.97734)
  MoveL 2220 to (222.27, 164.95, 41.04) mm, rotated rx -180 ry 0 rz 180 deg; joints [-69.319, 54.073, -69.461, 70.001, 95.378, 14.44]
  MoveL 2221 to (222.27, 164.95, 41.04) mm, rotated rx -180 ry 0 rz 180 deg; joints [-69.319, 54.073, -69.461, 70.001, 95.378, 14.44]
  Call Extruder(268.27004)
  MoveL 2222 to (221.68, 165, 41.04) mm, rotated rx 180 ry 0 rz 180 deg; joints [-69.504, 54.06, -69.467, 70.182, 95.338, 14.474]
  MoveL 2223 to (221.68, 165, 41.04) mm, rotated rx 180 ry 0 rz 180 deg; joints [-69.504, 54.06, -69.467, 70.182, 95.338, 14.474]
  Call Extruder(268.84349)
  MoveL 2224 to (220.52, 165.05, 41.04) mm, rotated rx 180 ry 0 rz -180 deg; joints [-69.864, 54.034, -69.481, 70.536, 95.261, 14.545]
  MoveL 2225 to (220.52, 165.05, 41.04) mm, rotated rx 180 ry 0 rz -180 deg; joints [-69.864, 54.034, -69.481, 70.536, 95.261, 14.545]
  Call Extruder(269.55750)
  MoveL 2226 to (219.06, 165.09, 41.03) mm, rotated rx 180 ry 0 rz 180 deg; joints [-70.315, 54, -69.499, 70.978, 95.165, 14.634]
  Call Extruder(386.40424)
  MoveL 2227 to (-19.06, 165.09, 41.04) mm, rotated rx -180 ry 0 rz 180 deg; joints [-137.325, 58.429, -65.978, 137.077, 84.457, 5.133]
  Call Extruder(386.83284)
  MoveL 2228 to (-19.94, 165.07, 41.04) mm, rotated rx -180 ry 0 rz 180 deg; joints [-137.467, 58.463, -65.936, 137.224, 84.5, 5.067]
  MoveL 2229 to (-19.94, 165.07, 41.04) mm, rotated rx -180 ry 0 rz 180 deg; joints [-137.467, 58.463, -65.936, 137.224, 84.5, 5.067]
  Call Extruder(387.40629)
  MoveL 2230 to (-21.1, 165.03, 41.04) mm, rotated rx -180 ry 0 rz -180 deg; joints [-137.659, 58.509, -65.882, 137.422, 84.557, 4.981]
  MoveL 2231 to (-21.1, 165.03, 41.04) mm, rotated rx -180 ry 0 rz -180 deg; joints [-137.659, 58.509, -65.882, 137.422, 84.557, 4.981]
  Call Extruder(387.84059)
  MoveL 2232 to (-21.97, 164.98, 41.03) mm, rotated rx 180 ry 0 rz 180 deg; joints [-137.804, 58.542, -65.842, 137.572, 84.599, 4.917]
  MoveL 2233 to (-21.97, 164.98, 41.03) mm, rotated rx 180 ry 0 rz 180 deg; joints [-137.804, 58.542, -65.842, 137.572, 84.599, 4.917]
  Call Extruder(388.13462)
  MoveL 2234 to (-22.56, 164.93, 41.04) mm, rotated rx -180 ry 0 rz 180 deg; joints [-137.905, 58.564, -65.815, 137.676, 84.626, 4.875]
  MoveL 2235 to (-22.56, 164.93, 41.04) mm, rotated rx -180 ry 0 rz 180 deg; joints [-137.905, 58.564, -65.815, 137.676, 84.626, 4.875]
  Call Extruder(388.42998)
  MoveL 2236 to (-23.15, 164.89, 41.04) mm, rotated rx -180 ry 0 rz 180 deg; joints [-138.004, 58.586, -65.788, 137.779, 84.654, 4.832]
  MoveL 2237 to (-23.15, 164.89, 41.04) mm, rotated rx -180 ry 0 rz 180 deg; joints [-138.004, 58.586, -65.788, 137.779, 84.654, 4.832]
  Call Extruder(388.67619)
  MoveL 2238 to (-23.64, 164.84, 41.04) mm, rotated rx -180 ry 0 rz 180 deg; joints [-138.088, 58.604, -65.766, 137.865, 84.677, 4.798]
  MoveL 2239 to (-23.64, 164.84, 41.04) mm, rotated rx -180 ry 0 rz 180 deg; joints [-138.088, 58.604, -65.766, 137.865, 84.677, 4.798]
  Call Extruder(388.87290)
  MoveL 2240 to (-24.03, 164.79, 41.04) mm, rotated rx 180 ry 0 rz 180 deg; joints [-138.156, 58.618, -65.749, 137.935, 84.694, 4.77]
  MoveL 2241 to (-24.03, 164.79, 41.04) mm, rotated rx 180 ry 0 rz 180 deg; joints [-138.156, 58.618, -65.749, 137.935, 84.694, 4.77]
  Call Extruder(389.07047)
  MoveL 2242 to (-24.42, 164.75, 41.04) mm, rotated rx 180 ry 0 rz 180 deg; joints [-138.224, 58.632, -65.732, 138.005, 84.712, 4.743]
  MoveL 2243 to (-24.42, 164.75, 41.04) mm, rotated rx 180 ry 0 rz 180 deg; joints [-138.224, 58.632, -65.732, 138.005, 84.712, 4.743]
  Call Extruder(389.26891)
  MoveL 2244 to (-24.8, 164.7, 41.03) mm, rotated rx -180 ry 0 rz 180 deg; joints [-138.292, 58.646, -65.714, 138.075, 84.729, 4.716]
  MoveL 2245 to (-24.8, 164.7, 41.03) mm, rotated rx -180 ry 0 rz 180 deg; joints [-138.292, 58.646, -65.714, 138.075, 84.729, 4.716]
  Call Extruder(389.46822)
  MoveL 2246 to (-25.19, 164.66, 41.04) mm, rotated rx -180 ry 0 rz 180 deg; joints [-138.359, 58.66, -65.697, 138.144, 84.747, 4.689]
  MoveL 2247 to (-25.19, 164.66, 41.04) mm, rotated rx -180 ry 0 rz 180 deg; joints [-138.359, 58.66, -65.697, 138.144, 84.747, 4.689]
  Call Extruder(389.62706)
  MoveL 2248 to (-25.5, 164.61, 41.04) mm, rotated rx -180 ry 0 rz 180 deg; joints [-138.415, 58.671, -65.684, 138.201, 84.76, 4.668]
  MoveL 2249 to (-25.5, 164.61, 41.04) mm, rotated rx -180 ry 0 rz 180 deg; joints [-138.415, 58.671, -65.684, 138.201, 84.76, 4.668]
  Call Extruder(389.78661)
  MoveL 2250 to (-25.8, 164.56, 41.04) mm, rotated rx -180 ry 0 rz 180 deg; joints [-138.47, 58.681, -65.671, 138.258, 84.773, 4.647]
  MoveL 2251 to (-25.8, 164.56, 41.04) mm, rotated rx -180 ry 0 rz 180 deg; joints [-138.47, 58.681, -65.671, 138.258, 84.773, 4.647]
  Call Extruder(389.94690)
  MoveL 2252 to (-26.11, 164.51, 41.04) mm, rotated rx 180 ry 0 rz 180 deg; joints [-138.525, 58.692, -65.658, 138.314, 84.786, 4.626]
  MoveL 2253 to (-26.11, 164.51, 41.04) mm, rotated rx 180 ry 0 rz 180 deg; joints [-138.525, 58.692, -65.658, 138.314, 84.786, 4.626]
  Call Extruder(390.10792)
  MoveL 2254 to (-26.41, 164.46, 41.04) mm, rotated rx -180 ry 0 rz -180 deg; joints [-138.58, 58.702, -65.645, 138.371, 84.8, 4.606]
  MoveL 2255 to (-26.41, 164.46, 41.04) mm, rotated rx -180 ry 0 rz -180 deg; joints [-138.58, 58.702, -65.645, 138.371, 84.8, 4.606]
  Call Extruder(390.26966)
  MoveL 2256 to (-26.72, 164.41, 41.04) mm, rotated rx -180 ry 0 rz -180 deg; joints [-138.635, 58.713, -65.631, 138.427, 84.813, 4.585]
  MoveL 2257 to (-26.72, 164.41, 41.04) mm, rotated rx -180 ry 0 rz -180 deg; joints [-138.635, 58.713, -65.631, 138.427, 84.813, 4.585]
  Call Extruder(390.43213)
  MoveL 2258 to (-27.03, 164.36, 41.04) mm, rotated rx -180 ry 0 rz 180 deg; joints [-138.69, 58.723, -65.618, 138.483, 84.826, 4.564]
  MoveL 2259 to (-27.03, 164.36, 41.04) mm, rotated rx -180 ry 0 rz 180 deg; joints [-138.69, 58.723, -65.618, 138.483, 84.826, 4.564]
  Call Extruder(390.56606)
  MoveL 2260 to (-27.27, 164.32, 41.04) mm, rotated rx -180 ry 0 rz 180 deg; joints [-138.736, 58.732, -65.608, 138.531, 84.837, 4.547]
  MoveL 2261 to (-27.27, 164.32, 41.04) mm, rotated rx -180 ry 0 rz 180 deg; joints [-138.736, 58.732, -65.608, 138.531, 84.837, 4.547]
  Call Extruder(390.70059)
  MoveL 2262 to (-27.52, 164.27, 41.04) mm, rotated rx -180 ry 0 rz 180 deg; joints [-138.783, 58.74, -65.597, 138.579, 84.847, 4.531]
  MoveL 2263 to (-27.52, 164.27, 41.04) mm, rotated rx -180 ry 0 rz 180 deg; joints [-138.783, 58.74, -65.597, 138.579, 84.847, 4.531]
  Call Extruder(390.83574)
  MoveL 2264 to (-27.77, 164.22, 41.04) mm, rotated rx -180 ry 0 rz -180 deg; joints [-138.829, 58.748, -65.587, 138.626, 84.857, 4.514]
  MoveL 2265 to (-27.77, 164.22, 41.04) mm, rotated rx -180 ry 0 rz -180 deg; joints [-138.829, 58.748, -65.587, 138.626, 84.857, 4.514]
  Call Extruder(390.97150)
  MoveL 2266 to (-28.02, 164.17, 41.04) mm, rotated rx -180 ry 0 rz 180 deg; joints [-138.875, 58.756, -65.576, 138.673, 84.868, 4.498]
  MoveL 2267 to (-28.02, 164.17, 41.04) mm, rotated rx -180 ry 0 rz 180 deg; joints [-138.875, 58.756, -65.576, 138.673, 84.868, 4.498]
  Call Extruder(391.10786)
  MoveL 2268 to (-28.27, 164.12, 41.04) mm, rotated rx -180 ry 0 rz 180 deg; joints [-138.921, 58.764, -65.566, 138.721, 84.878, 4.481]
  MoveL 2269 to (-28.27, 164.12, 41.04) mm, rotated rx -180 ry 0 rz 180 deg; joints [-138.921, 58.764, -65.566, 138.721, 84.878, 4.481]
  Call Extruder(391.24484)
  MoveL 2270 to (-28.52, 164.07, 41.04) mm, rotated rx -180 ry 0 rz -180 deg; joints [-138.967, 58.773, -65.555, 138.768, 84.889, 4.465]
  MoveL 2271 to (-28.52, 164.07, 41.04) mm, rotated rx -180 ry 0 rz -180 deg; joints [-138.967, 58.773, -65.555, 138.768, 84.889, 4.465]
  Call Extruder(391.38243)
  MoveL 2272 to (-28.77, 164.02, 41.04) mm, rotated rx 180 ry 0 rz -180 deg; joints [-139.013, 58.781, -65.545, 138.815, 84.899, 4.448]
  MoveL 2273 to (-28.77, 164.02, 41.04) mm, rotated rx 180 ry 0 rz -180 deg; joints [-139.013, 58.781, -65.545, 138.815, 84.899, 4.448]
  Call Extruder(391.49614)
  MoveL 2274 to (-28.97, 163.97, 41.04) mm, rotated rx 180 ry 0 rz 180 deg; joints [-139.052, 58.788, -65.536, 138.854, 84.908, 4.435]
  MoveL 2275 to (-28.97, 163.97, 41.04) mm, rotated rx 180 ry 0 rz 180 deg; joints [-139.052, 58.788, -65.536, 138.854, 84.908, 4.435]
  Call Extruder(391.61031)
  MoveL 2276 to (-29.18, 163.93, 41.04) mm, rotated rx -180 ry 0 rz 180 deg; joints [-139.09, 58.794, -65.528, 138.894, 84.916, 4.421]
  MoveL 2277 to (-29.18, 163.93, 41.04) mm, rotated rx -180 ry 0 rz 180 deg; joints [-139.09, 58.794, -65.528, 138.894, 84.916, 4.421]
  Call Extruder(391.72493)
  MoveL 2278 to (-29.38, 163.88, 41.04) mm, rotated rx -180 ry 0 rz -180 deg; joints [-139.128, 58.801, -65.519, 138.933, 84.925, 4.408]
  MoveL 2279 to (-29.38, 163.88, 41.04) mm, rotated rx -180 ry 0 rz -180 deg; joints [-139.128, 58.801, -65.519, 138.933, 84.925, 4.408]
  Call Extruder(391.84000)
  MoveL 2280 to (-29.59, 163.84, 41.04) mm, rotated rx 180 ry 0 rz 180 deg; joints [-139.166, 58.807, -65.511, 138.972, 84.933, 4.395]
  MoveL 2281 to (-29.59, 163.84, 41.04) mm, rotated rx 180 ry 0 rz 180 deg; joints [-139.166, 58.807, -65.511, 138.972, 84.933, 4.395]
  Call Extruder(391.96224)
  MoveL 2282 to (-29.8, 163.78, 41.04) mm, rotated rx -180 ry 0 rz 180 deg; joints [-139.208, 58.814, -65.502, 139.015, 84.941, 4.381]
  MoveL 2283 to (-29.8, 163.78, 41.04) mm, rotated rx -180 ry 0 rz 180 deg; joints [-139.208, 58.814, -65.502, 139.015, 84.941, 4.381]
  Call Extruder(392.09192)
  MoveL 2284 to (-30.02, 163.72, 41.03) mm, rotated rx 180 ry 0 rz 180 deg; joints [-139.253, 58.821, -65.494, 139.061, 84.949, 4.367]
  MoveL 2285 to (-30.02, 163.72, 41.03) mm, rotated rx 180 ry 0 rz 180 deg; joints [-139.253, 58.821, -65.494, 139.061, 84.949, 4.367]
  Call Extruder(392.22216)
  MoveL 2286 to (-30.25, 163.65, 41.04) mm, rotated rx -180 ry 0 rz 180 deg; joints [-139.298, 58.827, -65.485, 139.107, 84.957, 4.353]
  MoveL 2287 to (-30.25, 163.65, 41.04) mm, rotated rx -180 ry 0 rz 180 deg; joints [-139.298, 58.827, -65.485, 139.107, 84.957, 4.353]
  Call Extruder(392.35297)
  MoveL 2288 to (-30.47, 163.58, 41.04) mm, rotated rx -180 ry 0 rz 180 deg; joints [-139.343, 58.834, -65.477, 139.152, 84.965, 4.339]
  MoveL 2289 to (-30.47, 163.58, 41.04) mm, rotated rx -180 ry 0 rz 180 deg; joints [-139.343, 58.834, -65.477, 139.152, 84.965, 4.339]
  Call Extruder(392.48435)
  MoveL 2290 to (-30.7, 163.51, 41.04) mm, rotated rx -180 ry 0 rz 180 deg; joints [-139.388, 58.841, -65.468, 139.198, 84.973, 4.325]
  MoveL 2291 to (-30.7, 163.51, 41.04) mm, rotated rx -180 ry 0 rz 180 deg; joints [-139.388, 58.841, -65.468, 139.198, 84.973, 4.325]
  Call Extruder(392.59624)
  MoveL 2292 to (-30.88, 163.45, 41.04) mm, rotated rx -180 ry 0 rz -180 deg; joints [-139.427, 58.846, -65.461, 139.238, 84.98, 4.314]
  MoveL 2293 to (-30.88, 163.45, 41.04) mm, rotated rx -180 ry 0 rz -180 deg; joints [-139.427, 58.846, -65.461, 139.238, 84.98, 4.314]
  Call Extruder(392.70858)
  MoveL 2294 to (-31.07, 163.39, 41.04) mm, rotated rx -180 ry 0 rz -180 deg; joints [-139.465, 58.851, -65.454, 139.277, 84.987, 4.302]
  MoveL 2295 to (-31.07, 163.39, 41.04) mm, rotated rx -180 ry 0 rz -180 deg; joints [-139.465, 58.851, -65.454, 139.277, 84.987, 4.302]
  Call Extruder(392.82136)
  MoveL 2296 to (-31.26, 163.33, 41.03) mm, rotated rx 180 ry 0 rz 180 deg; joints [-139.504, 58.857, -65.447, 139.316, 84.993, 4.291]
  MoveL 2297 to (-31.26, 163.33, 41.03) mm, rotated rx 180 ry 0 rz 180 deg; joints [-139.504, 58.857, -65.447, 139.316, 84.993, 4.291]
  Call Extruder(392.93458)
  MoveL 2298 to (-31.45, 163.27, 41.04) mm, rotated rx -180 ry 0 rz -180 deg; joints [-139.542, 58.862, -65.44, 139.355, 85, 4.279]
  MoveL 2299 to (-31.45, 163.27, 41.04) mm, rotated rx -180 ry 0 rz -180 deg; joints [-139.542, 58.862, -65.44, 139.355, 85, 4.279]
  Call Extruder(393.04826)
  MoveL 2300 to (-31.64, 163.21, 41.04) mm, rotated rx -180 ry 0 rz 180 deg; joints [-139.581, 58.868, -65.433, 139.395, 85.006, 4.267]
  MoveL 2301 to (-31.64, 163.21, 41.04) mm, rotated rx -180 ry 0 rz 180 deg; joints [-139.581, 58.868, -65.433, 139.395, 85.006, 4.267]
  Call Extruder(393.23023)
  MoveL 2302 to (-31.93, 163.09, 41.04) mm, rotated rx 180 ry 0 rz 180 deg; joints [-139.645, 58.875, -65.423, 139.46, 85.015, 4.251]
  MoveL 2303 to (-31.93, 163.09, 41.04) mm, rotated rx 180 ry 0 rz 180 deg; joints [-139.645, 58.875, -65.423, 139.46, 85.015, 4.251]
  Call Extruder(393.41296)
  MoveL 2304 to (-32.22, 162.96, 41.04) mm, rotated rx -180 ry 0 rz 180 deg; joints [-139.709, 58.883, -65.413, 139.525, 85.023, 4.234]
  MoveL 2305 to (-32.22, 162.96, 41.04) mm, rotated rx -180 ry 0 rz 180 deg; joints [-139.709, 58.883, -65.413, 139.525, 85.023, 4.234]
  Call Extruder(393.58337)
  MoveL 2306 to (-32.49, 162.85, 41.04) mm, rotated rx 180 ry 0 rz -180 deg; joints [-139.768, 58.89, -65.404, 139.585, 85.031, 4.218]
  MoveL 2307 to (-32.49, 162.85, 41.04) mm, rotated rx 180 ry 0 rz -180 deg; joints [-139.768, 58.89, -65.404, 139.585, 85.031, 4.218]
  Call Extruder(393.74134)
  MoveL 2308 to (-32.74, 162.74, 41.04) mm, rotated rx 180 ry 0 rz 180 deg; joints [-139.823, 58.896, -65.396, 139.641, 85.038, 4.204]
  MoveL 2309 to (-32.74, 162.74, 41.04) mm, rotated rx 180 ry 0 rz 180 deg; joints [-139.823, 58.896, -65.396, 139.641, 85.038, 4.204]
  Call Extruder(393.89990)
  MoveL 2310 to (-32.99, 162.64, 41.04) mm, rotated rx -180 ry 0 rz 180 deg; joints [-139.878, 58.903, -65.387, 139.697, 85.046, 4.189]
  MoveL 2311 to (-32.99, 162.64, 41.04) mm, rotated rx -180 ry 0 rz 180 deg; joints [-139.878, 58.903, -65.387, 139.697, 85.046, 4.189]
  Call Extruder(394.10607)
  MoveL 2312 to (-33.29, 162.46, 41.04) mm, rotated rx 180 ry 0 rz 180 deg; joints [-139.953, 58.909, -65.379, 139.773, 85.051, 4.174]
  MoveL 2313 to (-33.29, 162.46, 41.04) mm, rotated rx 180 ry 0 rz 180 deg; joints [-139.953, 58.909, -65.379, 139.773, 85.051, 4.174]
  Call Extruder(394.31302)
  MoveL 2314 to (-33.6, 162.29, 41.04) mm, rotated rx -180 ry 0 rz 180 deg; joints [-140.028, 58.915, -65.371, 139.849, 85.057, 4.158]
  MoveL 2315 to (-33.6, 162.29, 41.04) mm, rotated rx -180 ry 0 rz 180 deg; joints [-140.028, 58.915, -65.371, 139.849, 85.057, 4.158]
  Call Extruder(394.52075)
  MoveL 2316 to (-33.9, 162.11, 41.04) mm, rotated rx 180 ry 0 rz -180 deg; joints [-140.103, 58.921, -65.363, 139.924, 85.063, 4.142]
  MoveL 2317 to (-33.9, 162.11, 41.04) mm, rotated rx 180 ry 0 rz -180 deg; joints [-140.103, 58.921, -65.363, 139.924, 85.063, 4.142]
  Call Extruder(394.72926)
  MoveL 2318 to (-34.21, 161.93, 41.04) mm, rotated rx -180 ry 0 rz 180 deg; joints [-140.178, 58.928, -65.354, 140, 85.068, 4.126]
  MoveL 2319 to (-34.21, 161.93, 41.04) mm, rotated rx -180 ry 0 rz 180 deg; joints [-140.178, 58.928, -65.354, 140, 85.068, 4.126]
  Call Extruder(394.90880)
  MoveL 2320 to (-34.45, 161.76, 41.04) mm, rotated rx -180 ry 0 rz -180 deg; joints [-140.244, 58.932, -65.349, 140.067, 85.071, 4.114]
  MoveL 2321 to (-34.45, 161.76, 41.04) mm, rotated rx -180 ry 0 rz -180 deg; joints [-140.244, 58.932, -65.349, 140.067, 85.071, 4.114]
  Call Extruder(395.24224)
  MoveL 2322 to (-34.9, 161.43, 41.04) mm, rotated rx 180 ry 0 rz 180 deg; joints [-140.366, 58.939, -65.34, 140.19, 85.075, 4.093]
  MoveL 2323 to (-34.9, 161.43, 41.04) mm, rotated rx 180 ry 0 rz 180 deg; joints [-140.366, 58.939, -65.34, 140.19, 85.075, 4.093]
  Call Extruder(395.57686)
  MoveL 2324 to (-35.35, 161.1, 41.04) mm, rotated rx 180 ry 0 rz -180 deg; joints [-140.489, 58.946, -65.33, 140.314, 85.079, 4.072]
  Call Extruder(396.40476)
  MoveL 2325 to (-36.39, 160.19, 41.04) mm, rotated rx 180 ry 0 rz 180 deg; joints [-140.797, 58.958, -65.315, 140.624, 85.078, 4.028]
  Call Extruder(397.03477)
  MoveL 2326 to (-37.09, 159.4, 41.04) mm, rotated rx -180 ry 0 rz -180 deg; joints [-141.034, 58.96, -65.311, 140.862, 85.066, 4.004]
  Call Extruder(397.38246)
  MoveL 2327 to (-37.45, 158.95, 41.04) mm, rotated rx -180 ry 0 rz 180 deg; joints [-141.165, 58.96, -65.312, 140.993, 85.056, 3.993]
  MoveL 2328 to (-37.45, 158.95, 41.04) mm, rotated rx -180 ry 0 rz 180 deg; joints [-141.165, 58.96, -65.312, 140.993, 85.056, 3.993]
  Call Extruder(397.68150)
  MoveL 2329 to (-37.75, 158.55, 41.04) mm, rotated rx -180 ry 0 rz 180 deg; joints [-141.278, 58.959, -65.313, 141.106, 85.046, 3.985]
  MoveL 2330 to (-37.75, 158.55, 41.04) mm, rotated rx -180 ry 0 rz 180 deg; joints [-141.278, 58.959, -65.313, 141.106, 85.046, 3.985]
  Call Extruder(397.80380)
  MoveL 2331 to (-37.87, 158.38, 41.04) mm, rotated rx 180 ry 0 rz 180 deg; joints [-141.324, 58.958, -65.314, 141.152, 85.042, 3.982]
  Set speed (130.0 mm/s)
  MoveL 2332 to (-39.5, 155.47, 41.04) mm, rotated rx 180 ry 0 rz -180 deg; joints [-142.07, 58.931, -65.35, 141.896, 84.941, 3.956]
  Call M_RunCode(106)
  MoveL 2333 to (-39.5, 155.47, 50.44) mm, rotated rx -180 ry 0 rz -180 deg; joints [-142.07, 60.351, -67.439, 141.857, 84.415, 4.371]
  MoveL 2334 to (-38.84, 156.79, 50.44) mm, rotated rx 180 ry 0 rz 180 deg; joints [-141.743, 60.367, -67.419, 141.531, 84.468, 4.38]
  Set speed (30.0 mm/s)
  MoveL 2335 to (-38.84, 156.79, 50.44) mm, rotated rx 180 ry 0 rz 180 deg; joints [-141.743, 60.367, -67.419, 141.531, 84.468, 4.38]
  Call Extruder(397.96209)
  MoveL 2336 to (-38.94, 156.54, 50.44) mm, rotated rx -180 ry 0 rz 180 deg; joints [-141.802, 60.363, -67.424, 141.59, 84.456, 4.38]
  MoveL 2337 to (-38.94, 156.54, 50.44) mm, rotated rx -180 ry 0 rz 180 deg; joints [-141.802, 60.363, -67.424, 141.59, 84.456, 4.38]
  Call Extruder(398.11977)
  MoveL 2338 to (-39.05, 156.29, 50.44) mm, rotated rx 180 ry 0 rz 180 deg; joints [-141.862, 60.359, -67.428, 141.649, 84.445, 4.38]
  MoveL 2339 to (-39.05, 156.29, 50.44) mm, rotated rx 180 ry 0 rz 180 deg; joints [-141.862, 60.359, -67.428, 141.649, 84.445, 4.38]
  Call Extruder(398.28986)
  MoveL 2340 to (-39.17, 156.02, 50.44) mm, rotated rx -180 ry 0 rz 180 deg; joints [-141.926, 60.355, -67.434, 141.713, 84.433, 4.379]
  MoveL 2341 to (-39.17, 156.02, 50.44) mm, rotated rx -180 ry 0 rz 180 deg; joints [-141.926, 60.355, -67.434, 141.713, 84.433, 4.379]
  Call Extruder(398.47220)
  MoveL 2342 to (-39.29, 155.73, 50.44) mm, rotated rx -180 ry 0 rz 180 deg; joints [-141.995, 60.35, -67.44, 141.781, 84.42, 4.379]
  MoveL 2343 to (-39.29, 155.73, 50.44) mm, rotated rx -180 ry 0 rz 180 deg; joints [-141.995, 60.35, -67.44, 141.781, 84.42, 4.379]
  Call Extruder(398.65378)
  MoveL 2344 to (-39.41, 155.44, 50.44) mm, rotated rx 180 ry 0 rz 180 deg; joints [-142.064, 60.346, -67.445, 141.85, 84.406, 4.378]
  MoveL 2345 to (-39.41, 155.44, 50.44) mm, rotated rx 180 ry 0 rz 180 deg; joints [-142.064, 60.346, -67.445, 141.85, 84.406, 4.378]
  Call Extruder(398.76724)
  MoveL 2346 to (-39.47, 155.25, 50.44) mm, rotated rx -180 ry 0 rz -180 deg; joints [-142.106, 60.342, -67.45, 141.891, 84.397, 4.379]
  MoveL 2347 to (-39.47, 155.25, 50.44) mm, rotated rx -180 ry 0 rz -180 deg; joints [-142.106, 60.342, -67.45, 141.891, 84.397, 4.379]
  Call Extruder(398.88025)
  MoveL 2348 to (-39.53, 155.06, 50.44) mm, rotated rx -180 ry 0 rz 180 deg; joints [-142.148, 60.339, -67.455, 141.933, 84.387, 4.38]
  MoveL 2349 to (-39.53, 155.06, 50.44) mm, rotated rx -180 ry 0 rz 180 deg; joints [-142.148, 60.339, -67.455, 141.933, 84.387, 4.38]
  Call Extruder(398.99282)
  MoveL 2350 to (-39.59, 154.87, 50.44) mm, rotated rx 180 ry 0 rz 180 deg; joints [-142.19, 60.335, -67.459, 141.975, 84.377, 4.381]
  MoveL 2351 to (-39.59, 154.87, 50.44) mm, rotated rx 180 ry 0 rz 180 deg; joints [-142.19, 60.335, -67.459, 141.975, 84.377, 4.381]
  Call Extruder(399.10494)
  MoveL 2352 to (-39.65, 154.68, 50.44) mm, rotated rx -180 ry 0 rz 180 deg; joints [-142.233, 60.332, -67.464, 142.017, 84.367, 4.382]
  MoveL 2353 to (-39.65, 154.68, 50.44) mm, rotated rx -180 ry 0 rz 180 deg; joints [-142.233, 60.332, -67.464, 142.017, 84.367, 4.382]
  Call Extruder(399.21662)
  MoveL 2354 to (-39.71, 154.49, 50.44) mm, rotated rx -180 ry 0 rz 180 deg; joints [-142.275, 60.328, -67.468, 142.059, 84.358, 4.383]
  MoveL 2355 to (-39.71, 154.49, 50.44) mm, rotated rx -180 ry 0 rz 180 deg; joints [-142.275, 60.328, -67.468, 142.059, 84.358, 4.383]
  Call Extruder(399.34770)
  MoveL 2356 to (-39.78, 154.27, 50.44) mm, rotated rx -180 ry 0 rz -180 deg; joints [-142.325, 60.323, -67.474, 142.108, 84.346, 4.384]
  MoveL 2357 to (-39.78, 154.27, 50.44) mm, rotated rx -180 ry 0 rz -180 deg; joints [-142.325, 60.323, -67.474, 142.108, 84.346, 4.384]
  Call Extruder(399.47821)
  MoveL 2358 to (-39.85, 154.05, 50.44) mm, rotated rx -180 ry 0 rz -180 deg; joints [-142.374, 60.319, -67.48, 142.157, 84.334, 4.386]
  MoveL 2359 to (-39.85, 154.05, 50.44) mm, rotated rx -180 ry 0 rz -180 deg; joints [-142.374, 60.319, -67.48, 142.157, 84.334, 4.386]
  Call Extruder(399.60815)
  MoveL 2360 to (-39.92, 153.82, 50.44) mm, rotated rx 180 ry 0 rz -180 deg; joints [-142.424, 60.315, -67.485, 142.206, 84.323, 4.387]
  MoveL 2361 to (-39.92, 153.82, 50.44) mm, rotated rx 180 ry 0 rz -180 deg; joints [-142.424, 60.315, -67.485, 142.206, 84.323, 4.387]
  Call Extruder(399.73753)
  MoveL 2362 to (-39.98, 153.6, 50.44) mm, rotated rx -180 ry 0 rz -180 deg; joints [-142.474, 60.31, -67.491, 142.255, 84.311, 4.388]
  MoveL 2363 to (-39.98, 153.6, 50.44) mm, rotated rx -180 ry 0 rz -180 deg; joints [-142.474, 60.31, -67.491, 142.255, 84.311, 4.388]
  Call Extruder(399.85951)
  MoveL 2364 to (-40.04, 153.39, 50.44) mm, rotated rx -180 ry 0 rz 180 deg; joints [-142.52, 60.306, -67.497, 142.301, 84.299, 4.39]
  MoveL 2365 to (-40.04, 153.39, 50.44) mm, rotated rx -180 ry 0 rz 180 deg; joints [-142.52, 60.306, -67.497, 142.301, 84.299, 4.39]
  Call Extruder(399.97437)
  MoveL 2366 to (-40.08, 153.18, 50.44) mm, rotated rx 180 ry 0 rz 180 deg; joints [-142.563, 60.301, -67.503, 142.343, 84.287, 4.393]
  MoveL 2367 to (-40.08, 153.18, 50.44) mm, rotated rx 180 ry 0 rz 180 deg; joints [-142.563, 60.301, -67.503, 142.343, 84.287, 4.393]
  Call Extruder(400.08877)
  MoveL 2368 to (-40.13, 152.98, 50.44) mm, rotated rx 180 ry 0 rz 180 deg; joints [-142.606, 60.296, -67.509, 142.386, 84.275, 4.395]
  MoveL 2369 to (-40.13, 152.98, 50.44) mm, rotated rx 180 ry 0 rz 180 deg; joints [-142.606, 60.296, -67.509, 142.386, 84.275, 4.395]
  Call Extruder(400.20273)
  MoveL 2370 to (-40.17, 152.77, 50.44) mm, rotated rx -180 ry 0 rz 180 deg; joints [-142.649, 60.291, -67.515, 142.429, 84.263, 4.397]
  MoveL 2371 to (-40.17, 152.77, 50.44) mm, rotated rx -180 ry 0 rz 180 deg; joints [-142.649, 60.291, -67.515, 142.429, 84.263, 4.397]
  Call Extruder(400.31623)
  MoveL 2372 to (-40.22, 152.57, 50.44) mm, rotated rx 180 ry 0 rz 180 deg; joints [-142.692, 60.286, -67.521, 142.471, 84.252, 4.4]
  MoveL 2373 to (-40.22, 152.57, 50.44) mm, rotated rx 180 ry 0 rz 180 deg; joints [-142.692, 60.286, -67.521, 142.471, 84.252, 4.4]
  Call Extruder(400.45351)
  MoveL 2374 to (-40.27, 152.32, 50.44) mm, rotated rx -180 ry 0 rz 180 deg; joints [-142.744, 60.28, -67.528, 142.522, 84.237, 4.403]
  MoveL 2375 to (-40.27, 152.32, 50.44) mm, rotated rx -180 ry 0 rz 180 deg; joints [-142.744, 60.28, -67.528, 142.522, 84.237, 4.403]
  Call Extruder(400.59019)
  MoveL 2376 to (-40.32, 152.07, 50.44) mm, rotated rx 180 ry 0 rz 180 deg; joints [-142.796, 60.274, -67.536, 142.574, 84.222, 4.406]
  MoveL 2377 to (-40.32, 152.07, 50.44) mm, rotated rx 180 ry 0 rz 180 deg; joints [-142.796, 60.274, -67.536, 142.574, 84.222, 4.406]
  Call Extruder(400.72625)
  MoveL 2378 to (-40.37, 151.82, 50.44) mm, rotated rx -180 ry 0 rz -180 deg; joints [-142.848, 60.268, -67.543, 142.625, 84.207, 4.409]
  MoveL 2379 to (-40.37, 151.82, 50.44) mm, rotated rx -180 ry 0 rz -180 deg; joints [-142.848, 60.268, -67.543, 142.625, 84.207, 4.409]
  Call Extruder(400.86170)
  MoveL 2380 to (-40.42, 151.57, 50.44) mm, rotated rx -180 ry 0 rz -180 deg; joints [-142.9, 60.262, -67.551, 142.676, 84.193, 4.412]
  MoveL 2381 to (-40.42, 151.57, 50.44) mm, rotated rx -180 ry 0 rz -180 deg; joints [-142.9, 60.262, -67.551, 142.676, 84.193, 4.412]
  Call Extruder(400.99654)
  MoveL 2382 to (-40.47, 151.32, 50.44) mm, rotated rx -180 ry 0 rz -180 deg; joints [-142.952, 60.256, -67.558, 142.728, 84.178, 4.414]
  MoveL 2383 to (-40.47, 151.32, 50.44) mm, rotated rx -180 ry 0 rz -180 deg; joints [-142.952, 60.256, -67.558, 142.728, 84.178, 4.414]
  Call Extruder(401.13077)
  MoveL 2384 to (-40.52, 151.07, 50.44) mm, rotated rx 180 ry 0 rz -180 deg; joints [-143.004, 60.251, -67.566, 142.779, 84.163, 4.417]
  MoveL 2385 to (-40.52, 151.07, 50.44) mm, rotated rx 180 ry 0 rz -180 deg; joints [-143.004, 60.251, -67.566, 142.779, 84.163, 4.417]
  Call Extruder(401.26438)
  MoveL 2386 to (-40.57, 150.82, 50.44) mm, rotated rx -180 ry 0 rz 180 deg; joints [-143.057, 60.245, -67.573, 142.831, 84.148, 4.42]
  MoveL 2387 to (-40.57, 150.82, 50.44) mm, rotated rx -180 ry 0 rz 180 deg; joints [-143.057, 60.245, -67.573, 142.831, 84.148, 4.42]
  Call Extruder(401.42647)
  MoveL 2388 to (-40.61, 150.52, 50.44) mm, rotated rx -180 ry 0 rz 180 deg; joints [-143.119, 60.237, -67.583, 142.892, 84.13, 4.424]
  MoveL 2389 to (-40.61, 150.52, 50.44) mm, rotated rx -180 ry 0 rz 180 deg; joints [-143.119, 60.237, -67.583, 142.892, 84.13, 4.424]
  Call Extruder(401.58783)
  MoveL 2390 to (-40.66, 150.21, 50.44) mm, rotated rx 180 ry 0 rz 180 deg; joints [-143.182, 60.229, -67.593, 142.954, 84.111, 4.429]
  MoveL 2391 to (-40.66, 150.21, 50.44) mm, rotated rx 180 ry 0 rz 180 deg; joints [-143.182, 60.229, -67.593, 142.954, 84.111, 4.429]
  Call Extruder(401.74847)
  MoveL 2392 to (-40.71, 149.91, 50.44) mm, rotated rx -180 ry 0 rz -180 deg; joints [-143.245, 60.221, -67.603, 143.016, 84.092, 4.433]
  MoveL 2393 to (-40.71, 149.91, 50.44) mm, rotated rx -180 ry 0 rz -180 deg; joints [-143.245, 60.221, -67.603, 143.016, 84.092, 4.433]
  Call Extruder(401.90837)
  MoveL 2394 to (-40.76, 149.6, 50.44) mm, rotated rx 180 ry 0 rz 180 deg; joints [-143.307, 60.213, -67.612, 143.077, 84.073, 4.437]
  MoveL 2395 to (-40.76, 149.6, 50.44) mm, rotated rx 180 ry 0 rz 180 deg; joints [-143.307, 60.213, -67.612, 143.077, 84.073, 4.437]
  Call Extruder(402.06755)
  MoveL 2396 to (-40.81, 149.3, 50.44) mm, rotated rx -180 ry 0 rz 180 deg; joints [-143.37, 60.205, -67.622, 143.139, 84.054, 4.441]
  MoveL 2397 to (-40.81, 149.3, 50.44) mm, rotated rx -180 ry 0 rz 180 deg; joints [-143.37, 60.205, -67.622, 143.139, 84.054, 4.441]
  Call Extruder(402.22600)
  MoveL 2398 to (-40.86, 148.99, 50.44) mm, rotated rx -180 ry 0 rz 180 deg; joints [-143.433, 60.198, -67.632, 143.201, 84.035, 4.445]
  MoveL 2399 to (-40.86, 148.99, 50.44) mm, rotated rx -180 ry 0 rz 180 deg; joints [-143.433, 60.198, -67.632, 143.201, 84.035, 4.445]
  Call Extruder(402.42488)
  MoveL 2400 to (-40.9, 148.6, 50.44) mm, rotated rx -180 ry 0 rz 180 deg; joints [-143.51, 60.187, -67.645, 143.277, 84.01, 4.451]
  MoveL 2401 to (-40.9, 148.6, 50.44) mm, rotated rx -180 ry 0 rz 180 deg; joints [-143.51, 60.187, -67.645, 143.277, 84.01, 4.451]
  Call Extruder(402.62289)
  MoveL 2402 to (-40.95, 148.22, 50.44) mm, rotated rx -180 ry 0 rz -180 deg; joints [-143.588, 60.177, -67.658, 143.354, 83.986, 4.457]
  MoveL 2403 to (-40.95, 148.22, 50.44) mm, rotated rx -180 ry 0 rz -180 deg; joints [-143.588, 60.177, -67.658, 143.354, 83.986, 4.457]
  Call Extruder(402.82003)
  MoveL 2404 to (-40.99, 147.83, 50.44) mm, rotated rx -180 ry 0 rz 180 deg; joints [-143.666, 60.166, -67.67, 143.43, 83.961, 4.463]
  MoveL 2405 to (-40.99, 147.83, 50.44) mm, rotated rx -180 ry 0 rz 180 deg; joints [-143.666, 60.166, -67.67, 143.43, 83.961, 4.463]
  Call Extruder(403.01630)
  MoveL 2406 to (-41.04, 147.44, 50.44) mm, rotated rx -180 ry 0 rz -180 deg; joints [-143.744, 60.156, -67.683, 143.507, 83.936, 4.469]
  MoveL 2407 to (-41.04, 147.44, 50.44) mm, rotated rx -180 ry 0 rz -180 deg; joints [-143.744, 60.156, -67.683, 143.507, 83.936, 4.469]
  Call Extruder(403.26199)
  MoveL 2408 to (-41.09, 146.95, 50.44) mm, rotated rx 180 ry 0 rz 180 deg; joints [-143.841, 60.142, -67.7, 143.602, 83.904, 4.477]
  MoveL 2409 to (-41.09, 146.95, 50.44) mm, rotated rx 180 ry 0 rz 180 deg; joints [-143.841, 60.142, -67.7, 143.602, 83.904, 4.477]
  Call Extruder(403.55672)
  MoveL 2410 to (-41.13, 146.36, 50.44) mm, rotated rx 180 ry 0 rz 180 deg; joints [-143.957, 60.125, -67.721, 143.716, 83.864, 4.487]
  MoveL 2411 to (-41.13, 146.36, 50.44) mm, rotated rx 180 ry 0 rz 180 deg; joints [-143.957, 60.125, -67.721, 143.716, 83.864, 4.487]
  Call Extruder(403.85012)
  MoveL 2412 to (-41.18, 145.77, 50.44) mm, rotated rx -180 ry 0 rz -180 deg; joints [-144.073, 60.108, -67.741, 143.83, 83.825, 4.496]
  MoveL 2413 to (-41.18, 145.77, 50.44) mm, rotated rx -180 ry 0 rz -180 deg; joints [-144.073, 60.108, -67.741, 143.83, 83.825, 4.496]
  Call Extruder(404.28345)
  MoveL 2414 to (-41.23, 144.9, 50.44) mm, rotated rx -180 ry 0 rz 180 deg; joints [-144.243, 60.082, -67.773, 143.997, 83.765, 4.512]
  MoveL 2415 to (-41.23, 144.9, 50.44) mm, rotated rx -180 ry 0 rz 180 deg; joints [-144.243, 60.082, -67.773, 143.997, 83.765, 4.512]
  Call Extruder(404.85561)
  MoveL 2416 to (-41.27, 143.74, 50.44) mm, rotated rx -180 ry 0 rz -180 deg; joints [-144.468, 60.046, -67.816, 144.217, 83.684, 4.533]
  MoveL 2417 to (-41.27, 143.74, 50.44) mm, rotated rx -180 ry 0 rz -180 deg; joints [-144.468, 60.046, -67.816, 144.217, 83.684, 4.533]
  Call Extruder(405.28344)
  MoveL 2418 to (-41.29, 142.86, 50.44) mm, rotated rx 180 ry 0 rz 180 deg; joints [-144.635, 60.019, -67.848, 144.382, 83.622, 4.55]
  Call Extruder(447.27697)
  MoveL 2419 to (-41.29, 57.14, 50.44) mm, rotated rx -180 ry 0 rz 180 deg; joints [-164.153, 57.726, -70.049, 163.798, 78.152, 3.414]
  MoveL 2420 to (-41.29, 57.14, 50.44) mm, rotated rx -180 ry 0 rz 180 deg; joints [-164.153, 57.726, -70.049, 163.798, 78.152, 3.414]
  Call Extruder(447.99254)
  MoveL 2421 to (-41.25, 55.68, 50.44) mm, rotated rx 180 ry 0 rz 180 deg; joints [-164.534, 57.697, -70.071, 164.184, 78.08, 3.348]
  MoveL 2422 to (-41.25, 55.68, 50.44) mm, rotated rx 180 ry 0 rz 180 deg; joints [-164.534, 57.697, -70.071, 164.184, 78.08, 3.348]
  Call Extruder(448.56728)
  MoveL 2423 to (-41.2, 54.52, 50.44) mm, rotated rx -180 ry 0 rz 180 deg; joints [-164.838, 57.673, -70.089, 164.493, 78.023, 3.295]
  MoveL 2424 to (-41.2, 54.52, 50.44) mm, rotated rx -180 ry 0 rz 180 deg; joints [-164.838, 57.673, -70.089, 164.493, 78.023, 3.295]
  Call Extruder(448.86068)
  MoveL 2425 to (-41.16, 53.93, 50.44) mm, rotated rx -180 ry 0 rz 180 deg; joints [-164.992, 57.66, -70.099, 164.648, 77.992, 3.269]
  MoveL 2426 to (-41.16, 53.93, 50.44) mm, rotated rx -180 ry 0 rz 180 deg; joints [-164.992, 57.66, -70.099, 164.648, 77.992, 3.269]
  Call Extruder(449.15541)
  MoveL 2427 to (-41.11, 53.34, 50.44) mm, rotated rx -180 ry 0 rz -180 deg; joints [-165.145, 57.647, -70.109, 164.803, 77.961, 3.243]
  MoveL 2428 to (-41.11, 53.34, 50.44) mm, rotated rx -180 ry 0 rz -180 deg; joints [-165.145, 57.647, -70.109, 164.803, 77.961, 3.243]
  Call Extruder(449.45147)
  MoveL 2429 to (-41.06, 52.75, 50.44) mm, rotated rx -180 ry 0 rz 180 deg; joints [-165.299, 57.634, -70.119, 164.959, 77.93, 3.216]
  MoveL 2430 to (-41.06, 52.75, 50.44) mm, rotated rx -180 ry 0 rz 180 deg; joints [-165.299, 57.634, -70.119, 164.959, 77.93, 3.216]
  Call Extruder(449.64774)
  MoveL 2431 to (-41.02, 52.37, 50.44) mm, rotated rx -180 ry 0 rz -180 deg; joints [-165.399, 57.624, -70.126, 165.06, 77.908, 3.199]
  MoveL 2432 to (-41.02, 52.37, 50.44) mm, rotated rx -180 ry 0 rz -180 deg; joints [-165.399, 57.624, -70.126, 165.06, 77.908, 3.199]
  Call Extruder(449.84488)
  MoveL 2433 to (-40.97, 51.98, 50.44) mm, rotated rx -180 ry 0 rz -180 deg; joints [-165.499, 57.615, -70.134, 165.162, 77.886, 3.182]
  MoveL 2434 to (-40.97, 51.98, 50.44) mm, rotated rx -180 ry 0 rz -180 deg; joints [-165.499, 57.615, -70.134, 165.162, 77.886, 3.182]
  Call Extruder(450.04289)
  MoveL 2435 to (-40.93, 51.59, 50.44) mm, rotated rx 180 ry 0 rz 180 deg; joints [-165.6, 57.605, -70.141, 165.263, 77.865, 3.165]
  MoveL 2436 to (-40.93, 51.59, 50.44) mm, rotated rx 180 ry 0 rz 180 deg; joints [-165.6, 57.605, -70.141, 165.263, 77.865, 3.165]
  Call Extruder(450.24176)
  MoveL 2437 to (-40.88, 51.2, 50.44) mm, rotated rx 180 ry 0 rz 180 deg; joints [-165.7, 57.596, -70.148, 165.365, 77.843, 3.148]
  MoveL 2438 to (-40.88, 51.2, 50.44) mm, rotated rx 180 ry 0 rz 180 deg; joints [-165.7, 57.596, -70.148, 165.365, 77.843, 3.148]
  Call Extruder(450.42084)
  MoveL 2439 to (-40.83, 50.86, 50.44) mm, rotated rx -180 ry 0 rz 180 deg; joints [-165.79, 57.587, -70.154, 165.456, 77.823, 3.132]
  MoveL 2440 to (-40.83, 50.86, 50.44) mm, rotated rx -180 ry 0 rz 180 deg; joints [-165.79, 57.587, -70.154, 165.456, 77.823, 3.132]
  Call Extruder(450.58002)
  MoveL 2441 to (-40.78, 50.55, 50.44) mm, rotated rx 180 ry 0 rz 180 deg; joints [-165.869, 57.579, -70.161, 165.535, 77.805, 3.119]
  MoveL 2442 to (-40.78, 50.55, 50.44) mm, rotated rx 180 ry 0 rz 180 deg; joints [-165.869, 57.579, -70.161, 165.535, 77.805, 3.119]
  Call Extruder(450.73993)
  MoveL 2443 to (-40.73, 50.24, 50.44) mm, rotated rx 180 ry 0 rz 180 deg; joints [-165.948, 57.571, -70.167, 165.615, 77.787, 3.106]
  MoveL 2444 to (-40.73, 50.24, 50.44) mm, rotated rx 180 ry 0 rz 180 deg; joints [-165.948, 57.571, -70.167, 165.615, 77.787, 3.106]
  Call Extruder(450.90057)
  MoveL 2445 to (-40.69, 49.94, 50.44) mm, rotated rx -180 ry 0 rz -180 deg; joints [-166.026, 57.563, -70.173, 165.695, 77.769, 3.092]
  MoveL 2446 to (-40.69, 49.94, 50.44) mm, rotated rx -180 ry 0 rz -180 deg; joints [-166.026, 57.563, -70.173, 165.695, 77.769, 3.092]
  Call Extruder(451.06193)
  MoveL 2447 to (-40.64, 49.63, 50.44) mm, rotated rx -180 ry 0 rz -180 deg; joints [-166.105, 57.555, -70.179, 165.775, 77.751, 3.079]
  MoveL 2448 to (-40.64, 49.63, 50.44) mm, rotated rx -180 ry 0 rz -180 deg; joints [-166.105, 57.555, -70.179, 165.775, 77.751, 3.079]
  Call Extruder(451.22402)
  MoveL 2449 to (-40.59, 49.33, 50.44) mm, rotated rx -180 ry 0 rz 180 deg; joints [-166.184, 57.546, -70.185, 165.855, 77.733, 3.065]
  MoveL 2450 to (-40.59, 49.33, 50.44) mm, rotated rx -180 ry 0 rz 180 deg; joints [-166.184, 57.546, -70.185, 165.855, 77.733, 3.065]
  Call Extruder(451.37222)
  MoveL 2451 to (-40.54, 49.05, 50.44) mm, rotated rx -180 ry 0 rz 180 deg; joints [-166.256, 57.539, -70.191, 165.927, 77.716, 3.053]
  MoveL 2452 to (-40.54, 49.05, 50.44) mm, rotated rx -180 ry 0 rz 180 deg; joints [-166.256, 57.539, -70.191, 165.927, 77.716, 3.053]
  Call Extruder(451.50645)
  MoveL 2453 to (-40.49, 48.8, 50.44) mm, rotated rx -180 ry 0 rz 180 deg; joints [-166.32, 57.532, -70.196, 165.992, 77.701, 3.042]
  MoveL 2454 to (-40.49, 48.8, 50.44) mm, rotated rx -180 ry 0 rz 180 deg; joints [-166.32, 57.532, -70.196, 165.992, 77.701, 3.042]
  Call Extruder(451.64129)
  MoveL 2455 to (-40.44, 48.55, 50.44) mm, rotated rx 180 ry 0 rz -180 deg; joints [-166.384, 57.524, -70.201, 166.057, 77.685, 3.031]
  MoveL 2456 to (-40.44, 48.55, 50.44) mm, rotated rx 180 ry 0 rz -180 deg; joints [-166.384, 57.524, -70.201, 166.057, 77.685, 3.031]
  Call Extruder(451.77674)
  MoveL 2457 to (-40.39, 48.3, 50.44) mm, rotated rx 180 ry 0 rz 180 deg; joints [-166.448, 57.517, -70.207, 166.121, 77.67, 3.02]
  MoveL 2458 to (-40.39, 48.3, 50.44) mm, rotated rx 180 ry 0 rz 180 deg; joints [-166.448, 57.517, -70.207, 166.121, 77.67, 3.02]
  Call Extruder(451.91280)
  MoveL 2459 to (-40.34, 48.05, 50.44) mm, rotated rx -180 ry 0 rz 180 deg; joints [-166.512, 57.51, -70.212, 166.186, 77.654, 3.009]
  MoveL 2460 to (-40.34, 48.05, 50.44) mm, rotated rx -180 ry 0 rz 180 deg; joints [-166.512, 57.51, -70.212, 166.186, 77.654, 3.009]
  Call Extruder(452.04947)
  MoveL 2461 to (-40.29, 47.8, 50.44) mm, rotated rx -180 ry 0 rz 180 deg; joints [-166.576, 57.503, -70.217, 166.252, 77.639, 2.998]
  MoveL 2462 to (-40.29, 47.8, 50.44) mm, rotated rx -180 ry 0 rz 180 deg; joints [-166.576, 57.503, -70.217, 166.252, 77.639, 2.998]
  Call Extruder(452.18675)
  MoveL 2463 to (-40.24, 47.55, 50.44) mm, rotated rx -180 ry 0 rz 180 deg; joints [-166.641, 57.496, -70.222, 166.317, 77.623, 2.987]
  MoveL 2464 to (-40.24, 47.55, 50.44) mm, rotated rx -180 ry 0 rz 180 deg; joints [-166.641, 57.496, -70.222, 166.317, 77.623, 2.987]
  Call Extruder(452.31242)
  MoveL 2465 to (-40.2, 47.33, 50.44) mm, rotated rx 180 ry 0 rz -180 deg; joints [-166.699, 57.489, -70.227, 166.375, 77.609, 2.977]
  MoveL 2466 to (-40.2, 47.33, 50.44) mm, rotated rx 180 ry 0 rz -180 deg; joints [-166.699, 57.489, -70.227, 166.375, 77.609, 2.977]
  Call Extruder(452.42638)
  MoveL 2467 to (-40.15, 47.12, 50.44) mm, rotated rx -180 ry 0 rz 180 deg; joints [-166.751, 57.483, -70.232, 166.429, 77.596, 2.968]
  MoveL 2468 to (-40.15, 47.12, 50.44) mm, rotated rx -180 ry 0 rz 180 deg; joints [-166.751, 57.483, -70.232, 166.429, 77.596, 2.968]
  Call Extruder(452.54078)
  MoveL 2469 to (-40.11, 46.92, 50.44) mm, rotated rx -180 ry 0 rz -180 deg; joints [-166.804, 57.477, -70.236, 166.482, 77.583, 2.959]
  MoveL 2470 to (-40.11, 46.92, 50.44) mm, rotated rx -180 ry 0 rz -180 deg; joints [-166.804, 57.477, -70.236, 166.482, 77.583, 2.959]
  Call Extruder(452.65564)
  MoveL 2471 to (-40.06, 46.72, 50.44) mm, rotated rx 180 ry 0 rz -180 deg; joints [-166.857, 57.471, -70.241, 166.535, 77.57, 2.95]
  MoveL 2472 to (-40.06, 46.72, 50.44) mm, rotated rx 180 ry 0 rz -180 deg; joints [-166.857, 57.471, -70.241, 166.535, 77.57, 2.95]
  Call Extruder(452.77095)
  MoveL 2473 to (-40.02, 46.51, 50.44) mm, rotated rx 180 ry 0 rz -180 deg; joints [-166.909, 57.465, -70.245, 166.588, 77.557, 2.941]
  MoveL 2474 to (-40.02, 46.51, 50.44) mm, rotated rx 180 ry 0 rz -180 deg; joints [-166.909, 57.465, -70.245, 166.588, 77.557, 2.941]
  Call Extruder(452.90034)
  MoveL 2475 to (-39.95, 46.29, 50.44) mm, rotated rx -180 ry 0 rz -180 deg; joints [-166.966, 57.457, -70.251, 166.646, 77.541, 2.932]
  MoveL 2476 to (-39.95, 46.29, 50.44) mm, rotated rx -180 ry 0 rz -180 deg; joints [-166.966, 57.457, -70.251, 166.646, 77.541, 2.932]
  Call Extruder(453.03028)
  MoveL 2477 to (-39.88, 46.06, 50.44) mm, rotated rx -180 ry 0 rz -180 deg; joints [-167.022, 57.449, -70.257, 166.703, 77.525, 2.923]
  MoveL 2478 to (-39.88, 46.06, 50.44) mm, rotated rx -180 ry 0 rz -180 deg; joints [-167.022, 57.449, -70.257, 166.703, 77.525, 2.923]
  Call Extruder(453.16079)
  MoveL 2479 to (-39.82, 45.84, 50.44) mm, rotated rx 180 ry 0 rz 180 deg; joints [-167.079, 57.441, -70.263, 166.76, 77.509, 2.913]
  MoveL 2480 to (-39.82, 45.84, 50.44) mm, rotated rx 180 ry 0 rz 180 deg; joints [-167.079, 57.441, -70.263, 166.76, 77.509, 2.913]
  Call Extruder(453.29187)
  MoveL 2481 to (-39.75, 45.62, 50.44) mm, rotated rx 180 ry 0 rz 180 deg; joints [-167.136, 57.433, -70.268, 166.817, 77.492, 2.904]
  MoveL 2482 to (-39.75, 45.62, 50.44) mm, rotated rx 180 ry 0 rz 180 deg; joints [-167.136, 57.433, -70.268, 166.817, 77.492, 2.904]
  Call Extruder(453.41351)
  MoveL 2483 to (-39.68, 45.41, 50.44) mm, rotated rx -180 ry 0 rz -180 deg; joints [-167.188, 57.426, -70.274, 166.87, 77.477, 2.895]
  MoveL 2484 to (-39.68, 45.41, 50.44) mm, rotated rx -180 ry 0 rz -180 deg; joints [-167.188, 57.426, -70.274, 166.87, 77.477, 2.895]
  Call Extruder(453.52564)
  MoveL 2485 to (-39.62, 45.22, 50.44) mm, rotated rx -180 ry 0 rz 180 deg; joints [-167.235, 57.419, -70.279, 166.918, 77.463, 2.888]
  MoveL 2486 to (-39.62, 45.22, 50.44) mm, rotated rx -180 ry 0 rz 180 deg; joints [-167.235, 57.419, -70.279, 166.918, 77.463, 2.888]
  Call Extruder(453.63821)
  MoveL 2487 to (-39.56, 45.03, 50.44) mm, rotated rx -180 ry 0 rz 180 deg; joints [-167.283, 57.412, -70.284, 166.967, 77.449, 2.88]
  MoveL 2488 to (-39.56, 45.03, 50.44) mm, rotated rx -180 ry 0 rz 180 deg; joints [-167.283, 57.412, -70.284, 166.967, 77.449, 2.88]
  Call Extruder(453.75122)
  MoveL 2489 to (-39.5, 44.85, 50.44) mm, rotated rx 180 ry 0 rz 180 deg; joints [-167.331, 57.405, -70.289, 167.015, 77.435, 2.872]
  MoveL 2490 to (-39.5, 44.85, 50.44) mm, rotated rx 180 ry 0 rz 180 deg; joints [-167.331, 57.405, -70.289, 167.015, 77.435, 2.872]
  Call Extruder(453.86468)
  MoveL 2491 to (-39.44, 44.66, 50.44) mm, rotated rx -180 ry 0 rz 180 deg; joints [-167.379, 57.398, -70.294, 167.063, 77.421, 2.864]
  MoveL 2492 to (-39.44, 44.66, 50.44) mm, rotated rx -180 ry 0 rz 180 deg; joints [-167.379, 57.398, -70.294, 167.063, 77.421, 2.864]
  Call Extruder(454.01232)
  MoveL 2493 to (-39.35, 44.42, 50.44) mm, rotated rx 180 ry 0 rz 180 deg; joints [-167.439, 57.389, -70.301, 167.124, 77.402, 2.854]
  MoveL 2494 to (-39.35, 44.42, 50.44) mm, rotated rx 180 ry 0 rz 180 deg; joints [-167.439, 57.389, -70.301, 167.124, 77.402, 2.854]
  Call Extruder(454.19466)
  MoveL 2495 to (-39.22, 44.12, 50.44) mm, rotated rx -180 ry 0 rz 180 deg; joints [-167.512, 57.377, -70.31, 167.197, 77.378, 2.843]
  MoveL 2496 to (-39.22, 44.12, 50.44) mm, rotated rx -180 ry 0 rz 180 deg; joints [-167.512, 57.377, -70.31, 167.197, 77.378, 2.843]
  Call Extruder(454.37775)
  MoveL 2497 to (-39.1, 43.83, 50.44) mm, rotated rx -180 ry 0 rz -180 deg; joints [-167.584, 57.364, -70.319, 167.271, 77.354, 2.831]
  MoveL 2498 to (-39.1, 43.83, 50.44) mm, rotated rx -180 ry 0 rz -180 deg; joints [-167.584, 57.364, -70.319, 167.271, 77.354, 2.831]
  Call Extruder(454.53544)
  MoveL 2499 to (-39, 43.58, 50.44) mm, rotated rx -180 ry 0 rz -180 deg; joints [-167.646, 57.354, -70.326, 167.333, 77.333, 2.822]
  MoveL 2500 to (-39, 43.58, 50.44) mm, rotated rx -180 ry 0 rz -180 deg; joints [-167.646, 57.354, -70.326, 167.333, 77.333, 2.822]
  Call Extruder(454.69372)
  MoveL 2501 to (-38.89, 43.34, 50.44) mm, rotated rx -180 ry 0 rz -180 deg; joints [-167.708, 57.343, -70.334, 167.396, 77.312, 2.812]
  MoveL 2502 to (-38.89, 43.34, 50.44) mm, rotated rx -180 ry 0 rz -180 deg; joints [-167.708, 57.343, -70.334, 167.396, 77.312, 2.812]
  Call Extruder(454.87574)
  MoveL 2503 to (-38.75, 43.06, 50.44) mm, rotated rx -180 ry 0 rz -180 deg; joints [-167.776, 57.329, -70.344, 167.464, 77.286, 2.802]
  MoveL 2504 to (-38.75, 43.06, 50.44) mm, rotated rx -180 ry 0 rz -180 deg; joints [-167.776, 57.329, -70.344, 167.464, 77.286, 2.802]
  Call Extruder(455.08230)
  MoveL 2505 to (-38.57, 42.75, 50.44) mm, rotated rx -180 ry 0 rz -180 deg; joints [-167.849, 57.313, -70.355, 167.538, 77.255, 2.791]
  MoveL 2506 to (-38.57, 42.75, 50.44) mm, rotated rx -180 ry 0 rz -180 deg; joints [-167.849, 57.313, -70.355, 167.538, 77.255, 2.791]
  Call Extruder(455.28963)
  MoveL 2507 to (-38.4, 42.45, 50.44) mm, rotated rx 180 ry 0 rz -180 deg; joints [-167.923, 57.297, -70.367, 167.612, 77.225, 2.781]
  MoveL 2508 to (-38.4, 42.45, 50.44) mm, rotated rx 180 ry 0 rz -180 deg; joints [-167.923, 57.297, -70.367, 167.612, 77.225, 2.781]
  Call Extruder(455.49774)
  MoveL 2509 to (-38.22, 42.15, 50.44) mm, rotated rx -180 ry 0 rz -180 deg; joints [-167.997, 57.281, -70.378, 167.686, 77.194, 2.77]
  MoveL 2510 to (-38.22, 42.15, 50.44) mm, rotated rx -180 ry 0 rz -180 deg; joints [-167.997, 57.281, -70.378, 167.686, 77.194, 2.77]
  Call Extruder(455.61546)
  MoveL 2511 to (-38.12, 41.98, 50.44) mm, rotated rx -180 ry 0 rz 180 deg; joints [-168.038, 57.272, -70.385, 167.727, 77.177, 2.764]
  MoveL 2512 to (-38.12, 41.98, 50.44) mm, rotated rx -180 ry 0 rz 180 deg; joints [-168.038, 57.272, -70.385, 167.727, 77.177, 2.764]
  Call Extruder(455.94830)
  MoveL 2513 to (-37.8, 41.52, 50.44) mm, rotated rx -180 ry 0 rz -180 deg; joints [-168.144, 57.244, -70.405, 167.834, 77.125, 2.75]
  MoveL 2514 to (-37.8, 41.52, 50.44) mm, rotated rx -180 ry 0 rz -180 deg; joints [-168.144, 57.244, -70.405, 167.834, 77.125, 2.75]
  Call Extruder(456.28234)
  MoveL 2515 to (-37.47, 41.07, 50.44) mm, rotated rx 180 ry 0 rz 180 deg; joints [-168.25, 57.215, -70.425, 167.94, 77.072, 2.737]
  MoveL 2516 to (-37.47, 41.07, 50.44) mm, rotated rx 180 ry 0 rz 180 deg; joints [-168.25, 57.215, -70.425, 167.94, 77.072, 2.737]
  Call Extruder(456.44993)
  MoveL 2517 to (-37.3, 40.85, 50.44) mm, rotated rx 180 ry 0 rz -180 deg; joints [-168.304, 57.201, -70.435, 167.994, 77.046, 2.729]
  Call Extruder(457.27924)
  MoveL 2518 to (-36.39, 39.81, 50.44) mm, rotated rx -180 ry 0 rz 180 deg; joints [-168.541, 57.125, -70.488, 168.231, 76.909, 2.702]
  Call Extruder(457.91031)
  MoveL 2519 to (-35.61, 39.11, 50.44) mm, rotated rx -180 ry 0 rz -180 deg; joints [-168.693, 57.062, -70.531, 168.382, 76.798, 2.689]
  MoveL 2520 to (-35.61, 39.11, 50.44) mm, rotated rx -180 ry 0 rz -180 deg; joints [-168.693, 57.062, -70.531, 168.382, 76.798, 2.689]
  Call Extruder(458.10788)
  MoveL 2521 to (-35.35, 38.9, 50.44) mm, rotated rx -180 ry 0 rz -180 deg; joints [-168.739, 57.042, -70.544, 168.428, 76.763, 2.685]
  Call Extruder(458.44190)
  MoveL 2522 to (-34.9, 38.57, 50.44) mm, rotated rx -180 ry 0 rz -180 deg; joints [-168.806, 57.007, -70.568, 168.494, 76.701, 2.681]
  MoveL 2523 to (-34.9, 38.57, 50.44) mm, rotated rx -180 ry 0 rz -180 deg; joints [-168.806, 57.007, -70.568, 168.494, 76.701, 2.681]
  Call Extruder(458.77473)
  MoveL 2524 to (-34.45, 38.24, 50.44) mm, rotated rx -180 ry 0 rz 180 deg; joints [-168.874, 56.972, -70.592, 168.561, 76.64, 2.677]
  MoveL 2525 to (-34.45, 38.24, 50.44) mm, rotated rx -180 ry 0 rz 180 deg; joints [-168.874, 56.972, -70.592, 168.561, 76.64, 2.677]
  Call Extruder(458.95398)
  MoveL 2526 to (-34.21, 38.07, 50.44) mm, rotated rx -180 ry 0 rz -180 deg; joints [-168.91, 56.953, -70.605, 168.596, 76.607, 2.675]
  MoveL 2527 to (-34.21, 38.07, 50.44) mm, rotated rx -180 ry 0 rz -180 deg; joints [-168.91, 56.953, -70.605, 168.596, 76.607, 2.675]
  Call Extruder(459.16208)
  MoveL 2528 to (-33.9, 37.89, 50.44) mm, rotated rx -180 ry 0 rz 180 deg; joints [-168.944, 56.93, -70.621, 168.629, 76.568, 2.675]
  MoveL 2529 to (-33.9, 37.89, 50.44) mm, rotated rx -180 ry 0 rz 180 deg; joints [-168.944, 56.93, -70.621, 168.629, 76.568, 2.675]
  Call Extruder(459.36942)
  MoveL 2530 to (-33.6, 37.71, 50.44) mm, rotated rx -180 ry 0 rz 180 deg; joints [-168.977, 56.906, -70.636, 168.661, 76.528, 2.675]
  MoveL 2531 to (-33.6, 37.71, 50.44) mm, rotated rx -180 ry 0 rz 180 deg; joints [-168.977, 56.906, -70.636, 168.661, 76.528, 2.675]
  Call Extruder(459.57597)
  MoveL 2532 to (-33.29, 37.54, 50.44) mm, rotated rx -180 ry 0 rz 180 deg; joints [-169.01, 56.883, -70.652, 168.693, 76.489, 2.675]
  MoveL 2533 to (-33.29, 37.54, 50.44) mm, rotated rx -180 ry 0 rz 180 deg; joints [-169.01, 56.883, -70.652, 168.693, 76.489, 2.675]
  Call Extruder(459.78174)
  MoveL 2534 to (-32.99, 37.36, 50.44) mm, rotated rx -180 ry 0 rz -180 deg; joints [-169.043, 56.86, -70.667, 168.725, 76.449, 2.674]
  MoveL 2535 to (-32.99, 37.36, 50.44) mm, rotated rx -180 ry 0 rz -180 deg; joints [-169.043, 56.86, -70.667, 168.725, 76.449, 2.674]
  Call Extruder(459.94004)
  MoveL 2536 to (-32.74, 37.26, 50.44) mm, rotated rx 180 ry 0 rz 180 deg; joints [-169.06, 56.841, -70.679, 168.741, 76.418, 2.677]
  MoveL 2537 to (-32.74, 37.26, 50.44) mm, rotated rx 180 ry 0 rz 180 deg; joints [-169.06, 56.841, -70.679, 168.741, 76.418, 2.677]
  Call Extruder(460.09774)
  MoveL 2538 to (-32.49, 37.15, 50.44) mm, rotated rx -180 ry 0 rz 180 deg; joints [-169.077, 56.823, -70.691, 168.757, 76.387, 2.679]
  MoveL 2539 to (-32.49, 37.15, 50.44) mm, rotated rx -180 ry 0 rz 180 deg; joints [-169.077, 56.823, -70.691, 168.757, 76.387, 2.679]
  Call Extruder(460.26783)
  MoveL 2540 to (-32.22, 37.03, 50.44) mm, rotated rx -180 ry 0 rz 180 deg; joints [-169.095, 56.802, -70.705, 168.774, 76.354, 2.681]
  MoveL 2541 to (-32.22, 37.03, 50.44) mm, rotated rx -180 ry 0 rz 180 deg; joints [-169.095, 56.802, -70.705, 168.774, 76.354, 2.681]
  Call Extruder(460.45016)
  MoveL 2542 to (-31.93, 36.91, 50.44) mm, rotated rx -180 ry 0 rz 180 deg; joints [-169.113, 56.781, -70.719, 168.791, 76.318, 2.684]
  MoveL 2543 to (-31.93, 36.91, 50.44) mm, rotated rx -180 ry 0 rz 180 deg; joints [-169.113, 56.781, -70.719, 168.791, 76.318, 2.684]
  Call Extruder(460.63174)
  MoveL 2544 to (-31.64, 36.79, 50.44) mm, rotated rx -180 ry 0 rz -180 deg; joints [-169.132, 56.759, -70.733, 168.809, 76.281, 2.686]
  MoveL 2545 to (-31.64, 36.79, 50.44) mm, rotated rx -180 ry 0 rz -180 deg; joints [-169.132, 56.759, -70.733, 168.809, 76.281, 2.686]
  Call Extruder(460.74519)
  MoveL 2546 to (-31.45, 36.73, 50.44) mm, rotated rx -180 ry 0 rz -180 deg; joints [-169.139, 56.745, -70.742, 168.815, 76.259, 2.689]
  MoveL 2547 to (-31.45, 36.73, 50.44) mm, rotated rx -180 ry 0 rz -180 deg; joints [-169.139, 56.745, -70.742, 168.815, 76.259, 2.689]
  Call Extruder(460.85821)
  MoveL 2548 to (-31.26, 36.67, 50.44) mm, rotated rx 180 ry 0 rz -180 deg; joints [-169.146, 56.731, -70.751, 168.821, 76.236, 2.692]
  MoveL 2549 to (-31.26, 36.67, 50.44) mm, rotated rx 180 ry 0 rz -180 deg; joints [-169.146, 56.731, -70.751, 168.821, 76.236, 2.692]
  Call Extruder(460.97078)
  MoveL 2550 to (-31.07, 36.61, 50.44) mm, rotated rx -180 ry 0 rz -180 deg; joints [-169.154, 56.717, -70.76, 168.828, 76.213, 2.695]
  MoveL 2551 to (-31.07, 36.61, 50.44) mm, rotated rx -180 ry 0 rz -180 deg; joints [-169.154, 56.717, -70.76, 168.828, 76.213, 2.695]
  Call Extruder(461.08290)
  MoveL 2552 to (-30.88, 36.55, 50.44) mm, rotated rx 180 ry 0 rz -180 deg; joints [-169.161, 56.703, -70.769, 168.834, 76.19, 2.698]
  MoveL 2553 to (-30.88, 36.55, 50.44) mm, rotated rx 180 ry 0 rz -180 deg; joints [-169.161, 56.703, -70.769, 168.834, 76.19, 2.698]
  Call Extruder(461.19458)
  MoveL 2554 to (-30.7, 36.49, 50.44) mm, rotated rx -180 ry 0 rz -180 deg; joints [-169.168, 56.689, -70.778, 168.841, 76.168, 2.7]
  MoveL 2555 to (-30.7, 36.49, 50.44) mm, rotated rx -180 ry 0 rz -180 deg; joints [-169.168, 56.689, -70.778, 168.841, 76.168, 2.7]
  Call Extruder(461.32566)
  MoveL 2556 to (-30.47, 36.42, 50.44) mm, rotated rx 180 ry 0 rz 180 deg; joints [-169.175, 56.673, -70.788, 168.847, 76.141, 2.704]
  MoveL 2557 to (-30.47, 36.42, 50.44) mm, rotated rx 180 ry 0 rz 180 deg; joints [-169.175, 56.673, -70.788, 168.847, 76.141, 2.704]
  Call Extruder(461.45616)
  MoveL 2558 to (-30.25, 36.35, 50.44) mm, rotated rx -180 ry 0 rz -180 deg; joints [-169.182, 56.656, -70.799, 168.853, 76.114, 2.708]
  MoveL 2559 to (-30.25, 36.35, 50.44) mm, rotated rx -180 ry 0 rz -180 deg; joints [-169.182, 56.656, -70.799, 168.853, 76.114, 2.708]
  Call Extruder(461.58611)
  MoveL 2560 to (-30.02, 36.28, 50.44) mm, rotated rx -180 ry 0 rz -180 deg; joints [-169.19, 56.64, -70.809, 168.859, 76.087, 2.711]
  MoveL 2561 to (-30.02, 36.28, 50.44) mm, rotated rx -180 ry 0 rz -180 deg; joints [-169.19, 56.64, -70.809, 168.859, 76.087, 2.711]
  Call Extruder(461.71549)
  MoveL 2562 to (-29.8, 36.22, 50.44) mm, rotated rx -180 ry 0 rz -180 deg; joints [-169.197, 56.623, -70.82, 168.865, 76.06, 2.715]
  MoveL 2563 to (-29.8, 36.22, 50.44) mm, rotated rx -180 ry 0 rz -180 deg; joints [-169.197, 56.623, -70.82, 168.865, 76.06, 2.715]
  Call Extruder(461.83745)
  MoveL 2564 to (-29.59, 36.16, 50.44) mm, rotated rx -180 ry 0 rz 180 deg; joints [-169.202, 56.608, -70.83, 168.869, 76.035, 2.719]
  MoveL 2565 to (-29.59, 36.16, 50.44) mm, rotated rx -180 ry 0 rz 180 deg; joints [-169.202, 56.608, -70.83, 168.869, 76.035, 2.719]
  Call Extruder(461.95230)
  MoveL 2566 to (-29.38, 36.12, 50.44) mm, rotated rx 180 ry 0 rz 180 deg; joints [-169.203, 56.593, -70.839, 168.869, 76.011, 2.723]
  MoveL 2567 to (-29.38, 36.12, 50.44) mm, rotated rx 180 ry 0 rz 180 deg; joints [-169.203, 56.593, -70.839, 168.869, 76.011, 2.723]
  Call Extruder(462.06669)
  MoveL 2568 to (-29.18, 36.07, 50.44) mm, rotated rx -180 ry 0 rz -180 deg; joints [-169.205, 56.578, -70.849, 168.87, 75.987, 2.727]
  MoveL 2569 to (-29.18, 36.07, 50.44) mm, rotated rx -180 ry 0 rz -180 deg; joints [-169.205, 56.578, -70.849, 168.87, 75.987, 2.727]
  Call Extruder(462.18063)
  MoveL 2570 to (-28.97, 36.03, 50.44) mm, rotated rx -180 ry 0 rz -180 deg; joints [-169.207, 56.563, -70.858, 168.87, 75.963, 2.732]
  MoveL 2571 to (-28.97, 36.03, 50.44) mm, rotated rx -180 ry 0 rz -180 deg; joints [-169.207, 56.563, -70.858, 168.87, 75.963, 2.732]
  Call Extruder(462.29412)
  MoveL 2572 to (-28.77, 35.98, 50.44) mm, rotated rx 180 ry 0 rz 180 deg; joints [-169.208, 56.548, -70.867, 168.871, 75.939, 2.736]
  MoveL 2573 to (-28.77, 35.98, 50.44) mm, rotated rx 180 ry 0 rz 180 deg; joints [-169.208, 56.548, -70.867, 168.871, 75.939, 2.736]
  Call Extruder(462.43141)
  MoveL 2574 to (-28.52, 35.93, 50.44) mm, rotated rx 180 ry 0 rz 180 deg; joints [-169.209, 56.53, -70.879, 168.87, 75.91, 2.742]
  MoveL 2575 to (-28.52, 35.93, 50.44) mm, rotated rx 180 ry 0 rz 180 deg; joints [-169.209, 56.53, -70.879, 168.87, 75.91, 2.742]
  Call Extruder(462.56808)
  MoveL 2576 to (-28.27, 35.88, 50.44) mm, rotated rx -180 ry 0 rz -180 deg; joints [-169.209, 56.512, -70.89, 168.869, 75.882, 2.748]
  MoveL 2577 to (-28.27, 35.88, 50.44) mm, rotated rx -180 ry 0 rz -180 deg; joints [-169.209, 56.512, -70.89, 168.869, 75.882, 2.748]
  Call Extruder(462.70414)
  MoveL 2578 to (-28.02, 35.83, 50.44) mm, rotated rx -180 ry 0 rz -180 deg; joints [-169.21, 56.494, -70.901, 168.868, 75.853, 2.753]
  MoveL 2579 to (-28.02, 35.83, 50.44) mm, rotated rx -180 ry 0 rz -180 deg; joints [-169.21, 56.494, -70.901, 168.868, 75.853, 2.753]
  Call Extruder(462.83959)
  MoveL 2580 to (-27.77, 35.78, 50.44) mm, rotated rx -180 ry 0 rz 180 deg; joints [-169.21, 56.476, -70.912, 168.867, 75.824, 2.759]
  MoveL 2581 to (-27.77, 35.78, 50.44) mm, rotated rx -180 ry 0 rz 180 deg; joints [-169.21, 56.476, -70.912, 168.867, 75.824, 2.759]
  Call Extruder(462.97443)
  MoveL 2582 to (-27.52, 35.73, 50.44) mm, rotated rx -180 ry 0 rz 180 deg; joints [-169.211, 56.457, -70.924, 168.867, 75.795, 2.765]
  MoveL 2583 to (-27.52, 35.73, 50.44) mm, rotated rx -180 ry 0 rz 180 deg; joints [-169.211, 56.457, -70.924, 168.867, 75.795, 2.765]
  Call Extruder(463.10867)
  MoveL 2584 to (-27.27, 35.68, 50.44) mm, rotated rx -180 ry 0 rz 180 deg; joints [-169.212, 56.439, -70.935, 168.866, 75.766, 2.771]
  MoveL 2585 to (-27.27, 35.68, 50.44) mm, rotated rx -180 ry 0 rz 180 deg; joints [-169.212, 56.439, -70.935, 168.866, 75.766, 2.771]
  Call Extruder(463.24229)
  MoveL 2586 to (-27.03, 35.63, 50.44) mm, rotated rx 180 ry 0 rz 180 deg; joints [-169.212, 56.421, -70.946, 168.865, 75.737, 2.776]
  MoveL 2587 to (-27.03, 35.63, 50.44) mm, rotated rx 180 ry 0 rz 180 deg; joints [-169.212, 56.421, -70.946, 168.865, 75.737, 2.776]
  Call Extruder(463.40438)
  MoveL 2588 to (-26.72, 35.59, 50.44) mm, rotated rx -180 ry 0 rz -180 deg; joints [-169.21, 56.399, -70.96, 168.86, 75.702, 2.784]
  MoveL 2589 to (-26.72, 35.59, 50.44) mm, rotated rx -180 ry 0 rz -180 deg; joints [-169.21, 56.399, -70.96, 168.86, 75.702, 2.784]
  Call Extruder(463.56576)
  MoveL 2590 to (-26.41, 35.54, 50.44) mm, rotated rx -180 ry 0 rz -180 deg; joints [-169.207, 56.376, -70.973, 168.856, 75.667, 2.792]
  MoveL 2591 to (-26.41, 35.54, 50.44) mm, rotated rx -180 ry 0 rz -180 deg; joints [-169.207, 56.376, -70.973, 168.856, 75.667, 2.792]
  Call Extruder(463.72640)
  MoveL 2592 to (-26.11, 35.49, 50.44) mm, rotated rx 180 ry 0 rz 180 deg; joints [-169.204, 56.354, -70.987, 168.851, 75.632, 2.8]
  MoveL 2593 to (-26.11, 35.49, 50.44) mm, rotated rx 180 ry 0 rz 180 deg; joints [-169.204, 56.354, -70.987, 168.851, 75.632, 2.8]
  Call Extruder(463.88631)
  MoveL 2594 to (-25.8, 35.44, 50.44) mm, rotated rx 180 ry 0 rz 180 deg; joints [-169.201, 56.332, -71, 168.846, 75.597, 2.808]
  MoveL 2595 to (-25.8, 35.44, 50.44) mm, rotated rx 180 ry 0 rz 180 deg; joints [-169.201, 56.332, -71, 168.846, 75.597, 2.808]
  Call Extruder(464.04550)
  MoveL 2596 to (-25.5, 35.39, 50.44) mm, rotated rx 180 ry 0 rz 180 deg; joints [-169.198, 56.309, -71.014, 168.841, 75.562, 2.816]
  MoveL 2597 to (-25.5, 35.39, 50.44) mm, rotated rx 180 ry 0 rz 180 deg; joints [-169.198, 56.309, -71.014, 168.841, 75.562, 2.816]
  Call Extruder(464.20396)
  MoveL 2598 to (-25.19, 35.34, 50.44) mm, rotated rx 180 ry 0 rz 180 deg; joints [-169.195, 56.287, -71.027, 168.836, 75.527, 2.824]
  MoveL 2599 to (-25.19, 35.34, 50.44) mm, rotated rx 180 ry 0 rz 180 deg; joints [-169.195, 56.287, -71.027, 168.836, 75.527, 2.824]
  Call Extruder(464.40284)
  MoveL 2600 to (-24.8, 35.3, 50.44) mm, rotated rx 180 ry 0 rz 180 deg; joints [-169.187, 56.259, -71.044, 168.825, 75.483, 2.835]
  MoveL 2601 to (-24.8, 35.3, 50.44) mm, rotated rx 180 ry 0 rz 180 deg; joints [-169.187, 56.259, -71.044, 168.825, 75.483, 2.835]
  Call Extruder(464.60085)
  MoveL 2602 to (-24.42, 35.25, 50.44) mm, rotated rx -180 ry 0 rz -180 deg; joints [-169.178, 56.231, -71.06, 168.815, 75.44, 2.846]
  MoveL 2603 to (-24.42, 35.25, 50.44) mm, rotated rx -180 ry 0 rz -180 deg; joints [-169.178, 56.231, -71.06, 168.815, 75.44, 2.846]
  Call Extruder(464.79799)
  MoveL 2604 to (-24.03, 35.21, 50.44) mm, rotated rx 180 ry 0 rz 180 deg; joints [-169.17, 56.202, -71.077, 168.804, 75.396, 2.857]
  MoveL 2605 to (-24.03, 35.21, 50.44) mm, rotated rx 180 ry 0 rz 180 deg; joints [-169.17, 56.202, -71.077, 168.804, 75.396, 2.857]
  Call Extruder(464.99426)
  MoveL 2606 to (-23.64, 35.16, 50.44) mm, rotated rx -180 ry 0 rz -180 deg; joints [-169.161, 56.174, -71.094, 168.793, 75.352, 2.868]
  MoveL 2607 to (-23.64, 35.16, 50.44) mm, rotated rx -180 ry 0 rz -180 deg; joints [-169.161, 56.174, -71.094, 168.793, 75.352, 2.868]
  Call Extruder(465.23995)
  MoveL 2608 to (-23.15, 35.11, 50.44) mm, rotated rx -180 ry 0 rz 180 deg; joints [-169.147, 56.138, -71.115, 168.775, 75.298, 2.883]
  MoveL 2609 to (-23.15, 35.11, 50.44) mm, rotated rx -180 ry 0 rz 180 deg; joints [-169.147, 56.138, -71.115, 168.775, 75.298, 2.883]
  Call Extruder(465.53467)
  MoveL 2610 to (-22.56, 35.07, 50.44) mm, rotated rx 180 ry 0 rz -180 deg; joints [-169.127, 56.095, -71.139, 168.751, 75.232, 2.902]
  MoveL 2611 to (-22.56, 35.07, 50.44) mm, rotated rx 180 ry 0 rz -180 deg; joints [-169.127, 56.095, -71.139, 168.751, 75.232, 2.902]
  Call Extruder(465.82807)
  MoveL 2612 to (-21.97, 35.02, 50.44) mm, rotated rx -180 ry 0 rz 180 deg; joints [-169.107, 56.052, -71.164, 168.726, 75.167, 2.921]
  MoveL 2613 to (-21.97, 35.02, 50.44) mm, rotated rx -180 ry 0 rz 180 deg; joints [-169.107, 56.052, -71.164, 168.726, 75.167, 2.921]
  Call Extruder(466.26140)
  MoveL 2614 to (-21.1, 34.97, 50.44) mm, rotated rx -180 ry 0 rz -180 deg; joints [-169.069, 55.989, -71.201, 168.682, 75.071, 2.952]
  MoveL 2615 to (-21.1, 34.97, 50.44) mm, rotated rx -180 ry 0 rz -180 deg; joints [-169.069, 55.989, -71.201, 168.682, 75.071, 2.952]
  Call Extruder(466.83356)
  MoveL 2616 to (-19.94, 34.93, 50.44) mm, rotated rx -180 ry 0 rz -180 deg; joints [-169.014, 55.904, -71.248, 168.618, 74.944, 2.993]
  MoveL 2617 to (-19.94, 34.93, 50.44) mm, rotated rx -180 ry 0 rz -180 deg; joints [-169.014, 55.904, -71.248, 168.618, 74.944, 2.993]
  Call Extruder(467.26139)
  MoveL 2618 to (-19.06, 34.91, 50.44) mm, rotated rx 180 ry 0 rz 180 deg; joints [-168.967, 55.84, -71.283, 168.565, 74.849, 3.026]
  Call Extruder(583.91008)
  MoveL 2619 to (219.06, 34.91, 50.44) mm, rotated rx -180 ry 0 rz 180 deg; joints [-30.588, 45.771, -73.468, 33.727, 113.586, 14.956]
  MoveL 2620 to (219.06, 34.91, 50.44) mm, rotated rx -180 ry 0 rz 180 deg; joints [-30.588, 45.771, -73.468, 33.727, 113.586, 14.956]
  Call Extruder(584.62565)
  MoveL 2621 to (220.52, 34.95, 50.44) mm, rotated rx 180 ry 0 rz 180 deg; joints [-30.009, 45.9, -73.471, 33.086, 113.628, 14.635]
  MoveL 2622 to (220.52, 34.95, 50.44) mm, rotated rx 180 ry 0 rz 180 deg; joints [-30.009, 45.9, -73.471, 33.086, 113.628, 14.635]
  Call Extruder(585.20039)
  MoveL 2623 to (221.68, 35, 50.44) mm, rotated rx -180 ry 0 rz 180 deg; joints [-29.572, 46.005, -73.473, 32.6, 113.651, 14.389]
  MoveL 2624 to (221.68, 35, 50.44) mm, rotated rx -180 ry 0 rz 180 deg; joints [-29.572, 46.005, -73.473, 32.6, 113.651, 14.389]
  Call Extruder(585.49378)
  MoveL 2625 to (222.27, 35.04, 50.44) mm, rotated rx -180 ry 0 rz 180 deg; joints [-29.371, 46.059, -73.473, 32.375, 113.656, 14.273]
  MoveL 2626 to (222.27, 35.04, 50.44) mm, rotated rx -180 ry 0 rz 180 deg; joints [-29.371, 46.059, -73.473, 32.375, 113.656, 14.273]
  Call Extruder(585.78851)
  MoveL 2627 to (222.86, 35.09, 50.44) mm, rotated rx -180 ry 0 rz 180 deg; joints [-29.173, 46.113, -73.474, 32.153, 113.659, 14.157]
  MoveL 2628 to (222.86, 35.09, 50.44) mm, rotated rx -180 ry 0 rz 180 deg; joints [-29.173, 46.113, -73.474, 32.153, 113.659, 14.157]
  Call Extruder(586.08457)
  MoveL 2629 to (223.45, 35.14, 50.44) mm, rotated rx -180 ry 0 rz -180 deg; joints [-28.978, 46.167, -73.475, 31.934, 113.661, 14.044]
  MoveL 2630 to (223.45, 35.14, 50.44) mm, rotated rx -180 ry 0 rz -180 deg; joints [-28.978, 46.167, -73.475, 31.934, 113.661, 14.044]
  Call Extruder(586.28084)
  MoveL 2631 to (223.83, 35.18, 50.44) mm, rotated rx -180 ry 0 rz 180 deg; joints [-28.862, 46.204, -73.475, 31.802, 113.659, 13.973]
  MoveL 2632 to (223.83, 35.18, 50.44) mm, rotated rx -180 ry 0 rz 180 deg; joints [-28.862, 46.204, -73.475, 31.802, 113.659, 13.973]
  Call Extruder(586.47798)
  MoveL 2633 to (224.22, 35.23, 50.44) mm, rotated rx 180 ry 0 rz 180 deg; joints [-28.747, 46.24, -73.475, 31.672, 113.656, 13.904]
  MoveL 2634 to (224.22, 35.23, 50.44) mm, rotated rx 180 ry 0 rz 180 deg; joints [-28.747, 46.24, -73.475, 31.672, 113.656, 13.904]
  Call Extruder(586.67599)
  MoveL 2635 to (224.61, 35.27, 50.44) mm, rotated rx -180 ry 0 rz 180 deg; joints [-28.633, 46.276, -73.475, 31.543, 113.652, 13.835]
  MoveL 2636 to (224.61, 35.27, 50.44) mm, rotated rx -180 ry 0 rz 180 deg; joints [-28.633, 46.276, -73.475, 31.543, 113.652, 13.835]
  Call Extruder(586.87487)
  MoveL 2637 to (225, 35.32, 50.44) mm, rotated rx 180 ry 0 rz 180 deg; joints [-28.52, 46.313, -73.476, 31.416, 113.648, 13.766]
  MoveL 2638 to (225, 35.32, 50.44) mm, rotated rx 180 ry 0 rz 180 deg; joints [-28.52, 46.313, -73.476, 31.416, 113.648, 13.766]
  Call Extruder(587.05395)
  MoveL 2639 to (225.34, 35.37, 50.44) mm, rotated rx -180 ry 0 rz -180 deg; joints [-28.425, 46.346, -73.476, 31.307, 113.643, 13.707]
  MoveL 2640 to (225.34, 35.37, 50.44) mm, rotated rx -180 ry 0 rz -180 deg; joints [-28.425, 46.346, -73.476, 31.307, 113.643, 13.707]
  Call Extruder(587.21313)
  MoveL 2641 to (225.65, 35.42, 50.44) mm, rotated rx -180 ry 0 rz 180 deg; joints [-28.346, 46.375, -73.476, 31.217, 113.637, 13.657]
  MoveL 2642 to (225.65, 35.42, 50.44) mm, rotated rx -180 ry 0 rz 180 deg; joints [-28.346, 46.375, -73.476, 31.217, 113.637, 13.657]
  Call Extruder(587.37304)
  MoveL 2643 to (225.96, 35.47, 50.44) mm, rotated rx 180 ry 0 rz 180 deg; joints [-28.267, 46.404, -73.476, 31.126, 113.63, 13.607]
  MoveL 2644 to (225.96, 35.47, 50.44) mm, rotated rx 180 ry 0 rz 180 deg; joints [-28.267, 46.404, -73.476, 31.126, 113.63, 13.607]
  Call Extruder(587.53368)
  MoveL 2645 to (226.26, 35.51, 50.44) mm, rotated rx 180 ry 0 rz 180 deg; joints [-28.19, 46.434, -73.476, 31.038, 113.623, 13.557]
  MoveL 2646 to (226.26, 35.51, 50.44) mm, rotated rx 180 ry 0 rz 180 deg; joints [-28.19, 46.434, -73.476, 31.038, 113.623, 13.557]
  Call Extruder(587.69505)
  MoveL 2647 to (226.57, 35.56, 50.44) mm, rotated rx 180 ry 0 rz 180 deg; joints [-28.112, 46.463, -73.476, 30.949, 113.616, 13.508]
  MoveL 2648 to (226.57, 35.56, 50.44) mm, rotated rx 180 ry 0 rz 180 deg; joints [-28.112, 46.463, -73.476, 30.949, 113.616, 13.508]
  Call Extruder(587.85714)
  MoveL 2649 to (226.87, 35.61, 50.44) mm, rotated rx -180 ry 0 rz 180 deg; joints [-28.036, 46.492, -73.476, 30.861, 113.609, 13.459]
  MoveL 2650 to (226.87, 35.61, 50.44) mm, rotated rx -180 ry 0 rz 180 deg; joints [-28.036, 46.492, -73.476, 30.861, 113.609, 13.459]
  Call Extruder(588.00405)
  MoveL 2651 to (227.15, 35.66, 50.44) mm, rotated rx -180 ry 0 rz -180 deg; joints [-27.971, 46.519, -73.476, 30.786, 113.601, 13.416]
  MoveL 2652 to (227.15, 35.66, 50.44) mm, rotated rx -180 ry 0 rz -180 deg; joints [-27.971, 46.519, -73.476, 30.786, 113.601, 13.416]
  Call Extruder(588.13568)
  MoveL 2653 to (227.39, 35.71, 50.44) mm, rotated rx -180 ry 0 rz -180 deg; joints [-27.917, 46.543, -73.476, 30.724, 113.593, 13.38]
  MoveL 2654 to (227.39, 35.71, 50.44) mm, rotated rx -180 ry 0 rz -180 deg; joints [-27.917, 46.543, -73.476, 30.724, 113.593, 13.38]
  Call Extruder(588.26790)
  MoveL 2655 to (227.64, 35.76, 50.44) mm, rotated rx -180 ry 0 rz -180 deg; joints [-27.863, 46.567, -73.475, 30.661, 113.585, 13.344]
  MoveL 2656 to (227.64, 35.76, 50.44) mm, rotated rx -180 ry 0 rz -180 deg; joints [-27.863, 46.567, -73.475, 30.661, 113.585, 13.344]
  Call Extruder(588.40071)
  MoveL 2657 to (227.88, 35.81, 50.44) mm, rotated rx 180 ry 0 rz 180 deg; joints [-27.81, 46.59, -73.475, 30.599, 113.576, 13.308]
  MoveL 2658 to (227.88, 35.81, 50.44) mm, rotated rx 180 ry 0 rz 180 deg; joints [-27.81, 46.59, -73.475, 30.599, 113.576, 13.308]
  Call Extruder(588.53410)
  MoveL 2659 to (228.12, 35.85, 50.44) mm, rotated rx -180 ry 0 rz 180 deg; joints [-27.758, 46.614, -73.475, 30.538, 113.568, 13.272]
  MoveL 2660 to (228.12, 35.85, 50.44) mm, rotated rx -180 ry 0 rz 180 deg; joints [-27.758, 46.614, -73.475, 30.538, 113.568, 13.272]
  Call Extruder(588.66808)
  MoveL 2661 to (228.37, 35.9, 50.44) mm, rotated rx 180 ry 0 rz 180 deg; joints [-27.705, 46.638, -73.475, 30.477, 113.559, 13.237]
  MoveL 2662 to (228.37, 35.9, 50.44) mm, rotated rx 180 ry 0 rz 180 deg; joints [-27.705, 46.638, -73.475, 30.477, 113.559, 13.237]
  Call Extruder(588.80265)
  MoveL 2663 to (228.61, 35.95, 50.44) mm, rotated rx 180 ry 0 rz 180 deg; joints [-27.653, 46.662, -73.475, 30.416, 113.55, 13.201]
  MoveL 2664 to (228.61, 35.95, 50.44) mm, rotated rx 180 ry 0 rz 180 deg; joints [-27.653, 46.662, -73.475, 30.416, 113.55, 13.201]
  Call Extruder(588.88871)
  MoveL 2665 to (228.77, 35.98, 50.44) mm, rotated rx -180 ry 0 rz 180 deg; joints [-27.619, 46.677, -73.475, 30.377, 113.545, 13.178]
  MoveL 2666 to (228.77, 35.98, 50.44) mm, rotated rx -180 ry 0 rz 180 deg; joints [-27.619, 46.677, -73.475, 30.377, 113.545, 13.178]
  Call Extruder(589.00224)
  MoveL 2667 to (228.97, 36.02, 50.44) mm, rotated rx -180 ry 0 rz 180 deg; joints [-27.575, 46.697, -73.474, 30.326, 113.537, 13.149]
  MoveL 2668 to (228.97, 36.02, 50.44) mm, rotated rx -180 ry 0 rz 180 deg; joints [-27.575, 46.697, -73.474, 30.326, 113.537, 13.149]
  Call Extruder(589.11625)
  MoveL 2669 to (229.18, 36.06, 50.44) mm, rotated rx -180 ry 0 rz 180 deg; joints [-27.531, 46.717, -73.474, 30.275, 113.53, 13.119]
  MoveL 2670 to (229.18, 36.06, 50.44) mm, rotated rx -180 ry 0 rz 180 deg; joints [-27.531, 46.717, -73.474, 30.275, 113.53, 13.119]
  Call Extruder(589.23074)
  MoveL 2671 to (229.38, 36.1, 50.44) mm, rotated rx -180 ry 0 rz 180 deg; joints [-27.487, 46.737, -73.474, 30.224, 113.523, 13.089]
  MoveL 2672 to (229.38, 36.1, 50.44) mm, rotated rx -180 ry 0 rz 180 deg; joints [-27.487, 46.737, -73.474, 30.224, 113.523, 13.089]
  Call Extruder(589.35620)
  MoveL 2673 to (229.6, 36.16, 50.44) mm, rotated rx -180 ry 0 rz 180 deg; joints [-27.455, 46.759, -73.474, 30.185, 113.51, 13.063]
